# B&R Automation Studio project PloterCNC (part 3)

```c
/*****************************************************************************/
/* BEGIN: fmi2SerializeFMUstate */
/*****************************************************************************/
fmi2Status fmi2SerializeFMUstate(fmi2Component		c,
								fmi2FMUstate		FMUstate,
								fmi2Byte 			serializedState[],
								size_t				size) {
	ModelInstance* comp = (ModelInstance *)c;
	M_INT *icur;

	if (invalidState(comp, "fmi2SerializeFMUstate", modelInitialized))
		return fmi2Error;

	icur = (M_INT *)FMUstate;
	if(icur[0]!=FMUStateID) {
		compLog(compEnv, comp->instanceName, fmi2Error, "error",
			"fmi2SerializedFMUstate: called with invalid FMUstate");
		return fmi2Error;
	}
	if(icur[1]>(M_INT)size) {
		compLog(compEnv, comp->instanceName, fmi2Error, "error",
			"fmi2SerializedFMUstate: called with size not sufficient to contain FMUstate");
		return fmi2Error;
	}
	memcpy(serializedState, FMUstate, size);

	return fmi2OK;
}
/* END: fmi2SerializeFMUstate */
/*****************************************************************************/

/*****************************************************************************/
/* BEGIN: fmi2DeSerializeFMUstate */
/*****************************************************************************/
fmi2Status fmi2DeSerializeFMUstate(	fmi2Component	c,
									const fmi2Byte	serializedState[],
									size_t			size,
									fmi2FMUstate	*FMUstate) {
	ModelInstance* comp = (ModelInstance *)c;
	M_INT *icur;

	if (invalidState(comp, "fmi2DeSerializeFMUstate", modelInitialized))
		return fmi2Error;

	icur = (M_INT *)serializedState;
	if(icur[0]!=FMUStateID) {
		compLog(compEnv, comp->instanceName, fmi2Error, "error",
			"fmi2DeSerializedFMUstate: called with serializedState not containing valid FMUstate");
		return fmi2Error;
	}
	if(icur[1]>(M_INT)size) {
		compLog(compEnv, comp->instanceName, fmi2Error, "error",
			"fmi2SerializedFMUstate: called with size not sufficient to contain serializedState");
		return fmi2Error;
	}
	FMUstate[0] = (fmi2FMUstate)comp->functions.allocateMemory(1,size);
	memcpy(*FMUstate, serializedState, size);

	return fmi2OK;
}
/* END: fmi2DeSerializeFMUstate */
/*****************************************************************************/

/*****************************************************************************/
/* BEGIN: fmi2GetDirectionalDerivative */
/*****************************************************************************/
fmi2Status fmi2GetDirectionalDerivative(	fmi2Component			c,
										const fmi2ValueReference	vUnknown_ref[],
										size_t						nUnknown,
										const fmi2ValueReference	vKnown_ref[],
										size_t						nKnown,
										const fmi2Real				dvKnown[],
										fmi2Real					dvUnknown[]) {
#ifdef FMI2_PROVIDES_DERIVATIVES
	int i, j, k, row, col, offset;
	fmi2Status sts;
	fmi2ValueReference vrs, vrd;
	ModelInstance* comp = (ModelInstance *)c;

	if (invalidState(comp, "fmi2GetDirectionalDerivatives", modelInstantiated|modelInitialized))
		return fmi2Error;
	if (nKnown>0 && nullPointer(comp, "fmi2GetDirectionalDerivative", "vKnown_ref[]", vKnown_ref))
		return fmi2Error;
	if (nUnknown>0 && nullPointer(comp, "fmi2GetDirectionalDerivative", "vUnknown_ref[]", vUnknown_ref))
		return fmi2Error;
	if (nKnown>0 && nullPointer(comp, "fmi2GetDirectionalDerivative", "dvKnown[]", dvKnown))
		return fmi2Error;

	sts = syncModel(comp,"fmi2GetDirectionalDerivative");
	if ( sts!=fmi2OK ) return sts;

	/* Initialize unknown vector */
	for (i=0; i<nUnknown; i++) dvUnknown[i] = 0.;

	/* Get Jacobian information, dimensions, data, etc? */
	if(!comp->jsynced) {
		if(comp->initializeMode)
			initjac(comp->S.w[0],&(comp->S.w[1]),&(comp->S.w[NEQ+NPAR+1]),comp->initRes,comp->initJacobian);
		else
			intjac(comp->S.w[0],&(comp->S.w[1]),&(comp->S.w[NEQ+NPAR+1]),comp->Jacobian);
		comp->jsynced = fmi2True;
	}

	/* Order of value references :
	t, #states, #index-1(inps), #discrete, #params, #derivs, #events */

	/* Start the computation loop */
	if (comp->initializeMode) {
		offset = NIKNO;
		for (i=0; i<nKnown; i++) {
			/* Check the seed */
			if (dvKnown[i]!=0) {
				vrs = vKnown_ref[i];
				/* assert(vr>=0 && vr<NUMBER_OF_REALS); */
				col = -1;
				for (k=0; k<NIKNO; k++)
					if (vrs==vrIknowns[k]) {
						col = k;
						break;
					}
				/* Compute column i */
				for (j=0; j<nUnknown; j++) {
					vrd = vUnknown_ref[j];
					/* assert(vrd>=0 && vrd<NUMBER_OF_REALS); */
					if ( vrd==vrs ) {
						dvUnknown[j] += 1.0;
					}
					else if(col!=-1) {
						for (k=0; k<NIUNK; k++)
							if (vrd==vrIunknowns[k]) {
								dvUnknown[j] += dvKnown[i]*comp->initJacobian[k*offset+col];
								break;
							}
					}
				}
			}
		}
	}
	else {
		offset = 1+NDIFF+NINP;
		for (i=0; i<nKnown; i++) {
			/* Check the seed */
			if (dvKnown[i]!=0) {
				vrs = vKnown_ref[i];
				/* assert(vr>=0 && vr<NUMBER_OF_REALS); */
				/* Check that vKnown_ref[i] is a state or input */
				if ( vrs==0 || (vrs>=vrStates[0] && vrs<vrStates[0]+NDIFF) )
					col = vrs;
				else if(vrs>=1+NDIFF+NIX1-NINP && vrs<1+NDIFF+NIX1)
					col = vrs-(NIX1-NINP);
				else
					return fmi2Error;
				/* Compute column i */
				for (j=0; j<nUnknown; j++) {
					vrd = vUnknown_ref[j];
					/* assert(vrd>=0 && vrd<NUMBER_OF_REALS); */
					/* Check if vrd is a derivative or an output,
					it could also be an output that's a state */
					if ( vrd>=vrDers[0] && vrd<vrDers[0]+NDIFF ) {
						row = vrd-vrDers[0];
						dvUnknown[j] += dvKnown[i]*comp->Jacobian[row*offset+col];
					}
					else if( vrd>=vrStates[0] && vrd<vrStates[0]+NDIFF ) {
						if ( vrd==vrs ) dvUnknown[j] += 1.0;
					}
					else {
						for (k=0; k<NOUT; k++)
							if (vrd==vrOuts[k]) {
								/* refval-t-states+derivs: vrd-1-NDIFF+NDIFF */
								row = vrd-1;
								dvUnknown[j] += dvKnown[i]*comp->Jacobian[row*offset+col];
								break;
							}
						if (k==NOUT) return fmi2Error;
					}
				}
			}
		}
	}
	return fmi2OK;
#else
	/* Compiler warning fix */
	int i=nUnknown+nKnown;
	void *tmp;
	tmp=(void *)vUnknown_ref;
	tmp=(void *)vKnown_ref;
	tmp=(void *)dvKnown;
	tmp=(void *)dvUnknown;
	if(i>0) tmp=(void *)c;
	/* End compiler warning fix */
	return fmi2Error;
#endif
}
/* END: fmi2GetDirectionalDerivative */
/*****************************************************************************/

#if NCON>0 && defined(WMI_PROJECTION)
/*****************************************************************************/
/* BEGIN: fmi2Projection */
/*****************************************************************************/
fmi2Status fmi2Projection(	fmi2Component	c,
								fmi2Real	P[],
								fmi2Real	projectionTolerance,
								size_t	iterationLimit,
								fmi2Boolean	apply) {
	int i;
	fmi2Status sts;
	fmi2Real S2[NDIFF];

	ModelInstance* comp = (ModelInstance *)c;

	if (invalidState(comp, "fmi2Projection", modelInstantiated|modelInitialized))
		return fmi2Error;

	sts = syncModel(comp,"fmi2Projection");
	if ( sts!=fmi2OK ) return sts;

	for(i=0;i<NDIFF;i++) S2[i] = comp->S.w[i+1];
	i=Projection(comp->S.w[0], &comp->S.w[1], projectionTolerance, iterationLimit, NULL, comp->S.psto);
	if( i!=0 ){
		/* Restore state */
		for(i=0;i<NDIFF;i++) comp->S.w[i+1]=S2[i];
		return fmi2Discard;
	}
	for(i=0;i<NDIFF;i++) P[i] = comp->S.w[i+1]-S2[i];

	if( !apply ){
		for(i=0;i<NDIFF;i++) comp->S.w[i+1]=S2[i];
	}

	return fmi2OK;
}
/* END: fmi2Projection */
/*****************************************************************************/

/*****************************************************************************/
/* BEGIN: fmi2ProjectionStep: No longer supported */
/*****************************************************************************/
fmi2Status fmi2ProjectionStep(	fmi2Component	c,
									fmi2Real	S[]) {
	UNUSED(c);
	UNUSED(S);
		return fmi2Error;
}
/* END: fmi2ProjectionStep */
/*****************************************************************************/

/*****************************************************************************/
/* BEGIN: fmi2Constraint */
/*****************************************************************************/
fmi2Status fmi2Constraint(	fmi2Component	c,
								fmi2Real	C[]) {
	int cb, cr, nblk;
	fmi2Real blkdata[2];
	fmi2Status sts;

	ModelInstance* comp = (ModelInstance *)c;

	if (invalidState(comp, "fmi2Constraint", modelInstantiated|modelInitialized))
		return fmi2Error;

	sts = syncModel(comp,"fmi2Constraint");
	if ( sts!=fmi2OK ) return sts;

	/* Iterate over Residual blocks */
	Rblkp(comp->S.w[0], &comp->S.w[1], blkdata, 0, 0);
	nblk = (int)(blkdata[0]);
	cr = 0;
	for(cb=1;cb<=nblk;cb++) {
		Rblkp(comp->S.w[0], &comp->S.w[1], &C[cr], cb, 3);
		Rblkp(comp->S.w[0], &comp->S.w[1], blkdata, cb, 1);
		cr += (int)(blkdata[0]);
	}

	return fmi2OK;
}
/* END: fmi2Constraint*/
/*****************************************************************************/

/*****************************************************************************/
/* BEGIN: fmi2ConstraintJacobian: No longer supported */
/*****************************************************************************/
fmi2Status fmi2ConstraintJacobian(	fmi2Component	c,
										fmi2Real	J[]) {

	/* If this function is required at some point, the code will need to be
	modified to fill in the ncon x ndiff Matrix using a sequence of calls to
	the block-based Jacobian. It is known that this will provide 0 entries
	for block dependencies on vars from a prior block, but this will only
	slow convergence of a newton approach, and be irrelevant when sufficiently
	close to the solution manifold */
	UNUSED(c);
	UNUSED(J);
		return fmi2Error;
}
/* END: fmi2ConstraintJacobian*/
/*****************************************************************************/
#endif

#ifdef FMI2_COSIMULATION
/*****************************************************************************
 * FMI functions: only for FMI Co-Simulation 2.0
 *****************************************************************************/
/*****************************************************************************/
/* BEGIN: fmi2SetRealInputDerivatives */
fmi2Status fmi2SetRealInputDerivatives(	fmi2Component			c,
										const fmi2ValueReference vr[],
										size_t					nvr,
										const fmi2Integer		order[],
										const fmi2Real			value[]) {
	ModelInstance* comp = (ModelInstance *)c;

	if (invalidState(comp, "fmi2SetRealInputDerivatives", modelInitialized))
		return fmi2Error;
	if (comp->loggingOn)
		compLog(compEnv, comp->instanceName, fmi2OK, "log",
				"fmi2SetRealInputDerivatives: nvr= %d", nvr);

	compLog(NULL, comp->instanceName, fmi2Error, "warning",
			"fmi2SetRealInputDerivatives: ignoring function call."
			" This model cannot interpolate inputs: canInterpolateInputs = \"fmi2False\"");

	return fmi2Warning;
}
/* END: fmi2SetRealInputDerivatives */
/*****************************************************************************/

/*****************************************************************************/
/* BEGIN: fmi2GetRealOutputDerivatives */
fmi2Status fmi2GetRealOutputDerivatives(fmi2Component			c,
										const fmi2ValueReference vr[],
										size_t					nvr,
										const fmi2Integer		order[],
										fmi2Real				value[]) {
	int i;
	ModelInstance* comp = (ModelInstance *)c;

	if (invalidState(comp, "fmi2GetRealOutputDerivatives", modelInitialized))
		return fmi2Error;
	if (comp->loggingOn)
		compLog(compEnv, comp->instanceName, fmi2OK, "log",
				"fmi2GetRealOutputDerivatives: nvr= %d",	nvr);

	compLog(NULL, comp->instanceName, fmi2Error, "warning",
			"fmi2GetRealOutputDerivatives: ignoring function call."
			" This model cannot compute derivatives of outputs: MaxOutputDerivativeOrder=\"0\"");

	for (i=0; i<(int)nvr; i++) value[i] = 0;

	return fmi2Warning;
}
/* END: fmi2GetRealOutputDerivatives */
/*****************************************************************************/

#define MAX_STEP  1.00000000000000000e-03

/*****************************************************************************/
/* BEGIN: fmi2DoStep */
fmi2Status fmi2DoStep(  fmi2Component	c,
						fmi2Real		currentCommunicationPoint,
						fmi2Real		communicationStepSize,
						fmi2Boolean		newStep) {

	ModelInstance* comp	= (ModelInstance *)c;
	int		i;
	double	h;
	int		n;	/* how many internal steps to perform for one fmi2DoStep */
	int		k, hasEvent;
#if NEVT>0
	M_INT *modes;
	double	prevEventIndicators[max(NEVT, 1)], eventIndicators[max(NEVT, 1)];
#endif

	if (invalidState(comp, "fmi2DoStep", modelInitialized)) return fmi2Error;

	if (comp->loggingOn)
		compLog(compEnv, comp->instanceName, fmi2OK, "log", "fmi2DoStep: "
				"currentCommunicationPoint = %g, "
				"communicationStepSize = %g, "
				"newStep = fmi2%s",
				currentCommunicationPoint, communicationStepSize, newStep ? "True" : "False");

	if (comp->stopTimeDefined && currentCommunicationPoint+communicationStepSize > comp->stopTime) {
		comp->state = modelError;
		return fmi2Error;
	}

	if(communicationStepSize==0) {
		n = 1;
		h = 0.0;
	}
	else {
		n = (int)floor((communicationStepSize-1e-12)/MAX_STEP)+1;
		h = communicationStepSize/n;
	}

#if NPAR>0
	if(pchange) {
		SolverInitialize(&(comp->S));
		pchange=0;
		if (errorOccured>0) {
			setVidError(comp,NULL);
			if (comp->fptr) {
				writeErrorToFile(comp->fptr,NULL);
				comp->fptr = NULL;
			}
			comp->state = modelTerminated;
			logMessage(comp, "fmi2DoStep", "error", fmi2Error);
			return fmi2Error;
		}
		else if(errorOccured<0) {
			logMessage(comp, "fmi2DoStep", "warning", fmi2Warning);
			errorOccured=0;
		}
	}
#endif

#if NEVT>0
	/* Run to get initial event indicators */
	eev(comp->S.w[0],&(comp->S.w[1]),&(comp->S.w[1]),prevEventIndicators);
	modes=comp->S.iw;
	ComputeEventIndicators(prevEventIndicators,&(comp->S.w[1]),modes,
		&modes[3*NEVT],&modes[2*NEVT],&modes[4*NEVT]);
#endif

	comp->S.w[0] = currentCommunicationPoint;
	/* break the step into n steps and do a step */
	for (k=0; k<n; k++) {
#if NUMBER_OF_REALS>0
		if (h>0.0) {
			EulerStep(h,&(comp->S));
			if (errorOccured>0) {
				setVidError(comp,NULL);
				if (comp->fptr) {
					writeErrorToFile(comp->fptr,NULL);
					comp->fptr = NULL;
				}
				comp->state = modelTerminated;
				logMessage(comp,"EulerStep","error", fmi2Error);
				return fmi2Error;
			}
			else if(errorOccured<0) {
				logMessage(comp, "EulerStep", "warning", fmi2Warning);
				errorOccured=0;
			}
		}

		SolverUpdate(&(comp->S),0,1);
		if (errorOccured>0) {
			setVidError(comp,NULL);
			if (comp->fptr) {
				writeErrorToFile(comp->fptr,NULL);
				comp->fptr = NULL;
			}
			errorOccured = 0;
			comp->state = modelTerminated;
			logMessage(comp, "fmi2DoStep", "error", fmi2Discard);
			return fmi2Discard;
		}
		else if(errorOccured<0) {
			logMessage(comp, "fmi2DoStep", "warning", fmi2Warning);
			errorOccured=0;
		}
		comp->synced = fmi2True;
		comp->jsynced = fmi2False;

		i=SolverProject(&(comp->S));
		if(i<0 || errorOccured==1) {
			setVidError(comp,NULL);
			if (comp->fptr) {
				writeErrorToFile(comp->fptr,NULL);
				comp->fptr = NULL;
			}
			errorOccured = 0;
			comp->state = modelTerminated;
			logMessage(comp, "fmi2DoStep", "error", fmi2Error);
			return fmi2Error;
		}
		else if(i>0 || errorOccured==2) {
			compLog(compEnv, comp->instanceName, fmi2OK, "log",
					"fmi2DoStep: model requested termination at t = %g",
					comp->S.w[0]);
			setVidError(comp,NULL);
			if (comp->fptr) {
				writeErrorToFile(comp->fptr,NULL);
				comp->fptr = NULL;
			}
			errorOccured = 0;
			comp->state = modelTerminated;
			logMessage(comp, "fmi2DoStep", "warning", fmi2Discard);
			return fmi2Discard;
		}
		else if(errorOccured<0) {
			logMessage(comp, "fmi2DoStep", "warning", fmi2Warning);
			errorOccured=0;
		}
#endif
		hasEvent = 0;

#if NEVT>0
		/* check for state event */
		eev(comp->S.w[0],&(comp->S.w[1]),&(comp->S.w[1]),eventIndicators);
		modes=comp->S.iw;
		ComputeEventIndicators(eventIndicators,&(comp->S.w[1]),modes,
			&modes[3*NEVT],&modes[2*NEVT],&modes[4*NEVT]);
		for (i=0; i<NEVT; i++) {
			if (eventIndicators[i] * prevEventIndicators[i] < 0) {
				hasEvent = 1;
				if (comp->loggingOn)
					compLog(compEnv, comp->instanceName, fmi2OK, "log",
							"fmi2DoStep: state event at %g, z%d crosses zero -%c-",
							comp->S.w[0], i, eventIndicators[i]<0 ? '\\' : '/');
			}
			prevEventIndicators[i] = eventIndicators[i];
		}

		if (hasEvent) {
			i = RunEvents(comp->S.w, comp->S.iw, 0, -1, EVTITER, comp->S.psto);
			if (i>0 || errorOccured==2) {
				compLog(compEnv, comp->instanceName, fmi2OK, "log",
					"fmi2DoStep: model requested termination at t = %g",
					comp->S.w[0]);
			}
			else if (i<0 || errorOccured>0) {
				logMessage(comp, "fmi2DoStep", "error", fmi2Error);
			}
			if (i || errorOccured>0) {
				setVidError(comp,NULL);
				if (comp->fptr) {
					writeErrorToFile(comp->fptr,NULL);
					comp->fptr = NULL;
				}
				errorOccured = 0;
				comp->state = modelTerminated;
				return fmi2Discard;
			}
			if(errorOccured<0) {
				logMessage(comp, "fmi2DoStep", "warning", fmi2Warning);
				errorOccured=0;
			}
		}
#endif

		SolverOutputs(&(comp->S));
	}

	comp->lastSuccessfulTime = currentCommunicationPoint + communicationStepSize;
	comp->vidsts = 2;
 	if (comp->fptr)
		fwrite(comp->S.w,sizeof(fmi2Real),NEQ+1,comp->fptr);

	return fmi2OK;
}
/* END: fmi2DoStep */
/*****************************************************************************/

/*****************************************************************************/
/* BEGIN: fmi2CancelStep */
fmi2Status fmi2CancelStep(fmi2Component c) {
	ModelInstance* comp = (ModelInstance *)c;

	if (invalidState(comp, "fmi2CancelStep", modelInitialized)) return fmi2Error;
	if (comp->loggingOn)
		compLog(compEnv, comp->instanceName, fmi2OK, "log", "fmi2CancelStep");

	compLog(NULL, comp->instanceName, fmi2Error, "error",
			"fmi2CancelStep: Can be called when fmi2DoStep returned fmi2Pending."
			" This is not the case.");
	comp->state = modelError;
	return fmi2Error;
}
/* END: fmi2CancelStep */
/*****************************************************************************/

/*****************************************************************************/
/* BEGIN: fmi2GetStatus */
fmi2Status fmi2GetStatus(	fmi2Component		c,
							const fmi2StatusKind s,
							fmi2Status*			value) {
	ModelInstance* comp = (ModelInstance *)c;

	if (invalidState(comp, "fmi2GetStatus", modelInstantiated|modelInitialized))
		return fmi2Error;

	if (s==fmi2DoStepStatus) {
		if (comp->loggingOn) {
			compLog(compEnv, comp->instanceName, fmi2OK, "log",
				"[fmi2GetStatus]: fmi2StatusKind = fmi2DoStepStatus");
			compLog(NULL, comp->instanceName, fmi2Error, "error",
				"[fmi2GetStatus]: Can be called with fmi2DoStepStatus when fmi2DoStep returned fmi2Pending."
				" This is not the case.");
		}
		return fmi2Discard;
	}
	else
		return fmi2Discard;
}
/* END: fmi2GetStatus */
/*****************************************************************************/

/*****************************************************************************/
/* BEGIN: fmi2GetRealStatus */
fmi2Status fmi2GetRealStatus(	fmi2Component		c,
								const fmi2StatusKind s,
								fmi2Real*			value) {
	ModelInstance* comp = (ModelInstance *)c;

	if (invalidState(comp, "fmi2GetRealStatus", modelInstantiated|modelInitialized))
		return fmi2Discard;

	if (s==fmi2LastSuccessfulTime) {
		if (comp->loggingOn) {
			compLog(compEnv, comp->instanceName, fmi2OK, "log",
				"[fmi2GetRealStatus]: fmi2StatusKind = fmi2LastSuccessfulTime");
		}
		if (comp->state==modelTerminated) {
			*value = comp->lastSuccessfulTime;
			return fmi2OK;
		}
		else {
			compLog(NULL, comp->instanceName, fmi2Error, "error",
				"[fmi2GetRealStatus]: Can be called with fmi2LastSuccessfulTime when fmi2DoStep returned fmi2Discard."
				" This is not the case.");
			return fmi2Discard;
		}
	}
	else
		return fmi2Discard;
}
/* END: fmi2GetRealStatus */
/*****************************************************************************/

/*****************************************************************************/
/* BEGIN: fmi2GetIntegerStatus */
fmi2Status fmi2GetIntegerStatus(fmi2Component		c,
								const fmi2StatusKind s,
								fmi2Integer*		value) {
	return fmi2Discard;
}
/* END: fmi2GetIntegerStatus */
/*****************************************************************************/

/*****************************************************************************/
/* BEGIN: fmi2GetBooleanStatus */
fmi2Status fmi2GetBooleanStatus(fmi2Component		c,
								const fmi2StatusKind s,
								fmi2Boolean*		value) {
	ModelInstance* comp = (ModelInstance *)c;

	if (invalidState(comp, "fmi2GetBooleanStatus", modelInstantiated|modelInitialized))
		return fmi2Discard;

	if (s==fmi2Terminated) {
		if (comp->loggingOn) {
			compLog(compEnv, comp->instanceName, fmi2OK, "log",
				"[fmi2GetBooleanStatus]: fmi2StatusKind = fmi2Terminated");
		}
		if (comp->state==modelTerminated)
			*value = fmi2True;
		else
			*value = fmi2False;
		return fmi2OK;
	}
	else
		return fmi2Discard;
}
/* END: fmi2GetBooleanStatus */
/*****************************************************************************/

/*****************************************************************************/
/* BEGIN: fmi2GetStringStatus */
fmi2Status fmi2GetStringStatus(	fmi2Component		c,
								const fmi2StatusKind s,
								fmi2String*			value) {
	ModelInstance* comp = (ModelInstance *)c;

	if (invalidState(comp, "fmi2GetStringStatus", modelInstantiated|modelInitialized))
		return fmi2Discard;

	if (s==fmi2PendingStatus) {
		if (comp->loggingOn) {
			compLog(compEnv, comp->instanceName, fmi2OK, "log",
				"[fmi2GetStringStatus]: fmi2StatusKind = fmi2PendingStatus");
			compLog(NULL, comp->instanceName, fmi2Error, "error",
					"[fmi2GetStringStatus]: Can be called with fmi2PendingStatus when fmi2DoStep returned fmi2Pending."
					" This is not the case.");
		}
		return fmi2Discard;
	}
	else
		return fmi2Discard;
}
/* END: fmi2GetStringStatus */
/*****************************************************************************/

#else
/*****************************************************************************
 * FMI functions: only for Model Exchange 2.0
 *****************************************************************************/

/*****************************************************************************/
/* BEGIN: fmi2EnterEventMode */
fmi2Status fmi2EnterEventMode(fmi2Component c) {
	ModelInstance* comp = (ModelInstance *)c;

	if (comp) {
		comp->lastEventTime = comp->S.w[0]-1.0;
		return fmi2OK;
	}
	else
		return fmi2Error;
}
/* END: fmi2EnterEventMode */
/*****************************************************************************/

/*****************************************************************************/
/* BEGIN: fmi2NewDiscreteStates */
fmi2Status fmi2NewDiscreteStates(fmi2Component	c,
								fmi2EventInfo*	eventInfo) {
	ModelInstance* comp = (ModelInstance *)c;
	int i;
#if NEVT+NCON>0
	fmi2Real save[NEQ],val;
#endif
	if (invalidState(comp, "fmi2NewDiscreteStates", modelInitialized))
		return fmi2Error;
	if (nullPointer (comp, "fmi2NewDiscreteStates", "eventInfo", eventInfo))
		return fmi2Error;

	eventInfo->newDiscreteStatesNeeded				= fmi2False;
	eventInfo->nominalsOfContinuousStatesChanged	= fmi2False;
	eventInfo->valuesOfContinuousStatesChanged		= fmi2False;
	eventInfo->terminateSimulation					= fmi2False;
	eventInfo->nextEventTimeDefined					= fmi2False;
	eventInfo->nextEventTime						= -0.0;

#if NEVT+NCON>0
	for(i=0;i<NEQ;i++) save[i]=comp->S.w[i+1];
#endif
	i=SolverProject(&(comp->S));
	if (i<0 || errorOccured==1) {
		setVidError(comp,NULL);
		if (comp->fptr) {
			writeErrorToFile(comp->fptr,NULL);
			comp->fptr = NULL;
		}
		eventInfo->terminateSimulation = fmi2True;
		comp->state = modelTerminated;
		logMessage(comp, "fmi2NewDiscreteStates", "error", fmi2Error);
		return fmi2Error;
	}
	else if (i>0 || errorOccured==2) {
		compLog(compEnv, comp->instanceName, fmi2OK, "log",
				"fmi2NewDiscreteStates: model requested termination at t = %g",
				comp->S.w[0]);
		setVidError(comp,NULL);
		if (comp->fptr) {
			writeErrorToFile(comp->fptr,NULL);
			comp->fptr = NULL;
		}
		eventInfo->terminateSimulation = fmi2True;
		comp->state = modelTerminated;
		logMessage(comp, "fmi2NewDiscreteStates", "warning", fmi2Discard);
		return fmi2OK;
	}
	else if(errorOccured<0) {
		logMessage(comp, "fmi2NewDiscreteStates", "warning", fmi2Warning);
		errorOccured=0;
	}
#if NEVT>0
	if (comp->S.w[0]!=comp->lastEventTime) {
		i=RunEvents(comp->S.w, comp->S.iw, 0, -1, EVTITER, comp->S.psto);
		if (i<0 || errorOccured==1) {
			setVidError(comp,NULL);
			if (comp->fptr) {
				writeErrorToFile(comp->fptr,NULL);
				comp->fptr = NULL;
			}
			eventInfo->terminateSimulation = fmi2True;
			comp->state = modelTerminated;
			logMessage(comp, "fmi2NewDiscreteStates", "error", fmi2Error);
			return fmi2Error;
		}
		else if (i>0 || errorOccured==2) {
			compLog(compEnv, comp->instanceName, fmi2OK, "log",
					"fmi2NewDiscreteStates: model requested termination at t = %g",
					comp->S.w[0]);
			setVidError(comp,NULL);
			if (comp->fptr) {
				writeErrorToFile(comp->fptr,NULL);
				comp->fptr = NULL;
			}
			eventInfo->terminateSimulation = fmi2True;
			comp->state = modelTerminated;
			logMessage(comp, "fmi2NewDiscreteStates", "warning", fmi2Discard);
			return fmi2OK;
		}
		else if(errorOccured<0) {
			logMessage(comp, "fmi2NewDiscreteStates", "warning", fmi2Warning);
			errorOccured=0;
		}
		comp->lastEventTime = comp->S.w[0];
	}
	i=RunEvents(comp->S.w, comp->S.iw, 1, -1, EVTITER, comp->S.psto);
	if (i<0 || errorOccured==1) {
		setVidError(comp,NULL);
		if (comp->fptr) {
			writeErrorToFile(comp->fptr,NULL);
			comp->fptr = NULL;
		}
		eventInfo->terminateSimulation = fmi2True;
		comp->state = modelTerminated;
		logMessage(comp, "fmi2NewDiscreteStates", "error", fmi2Error);
		return fmi2Error;
	}
	else if (i>0 || errorOccured==2) {
		compLog(compEnv, comp->instanceName, fmi2OK, "log",
				"fmi2NewDiscreteStates: model requested termination at t = %g",
				comp->S.w[0]);
		setVidError(comp,NULL);
		if (comp->fptr) {
			writeErrorToFile(comp->fptr,NULL);
			comp->fptr = NULL;
		}
		eventInfo->terminateSimulation = fmi2True;
		comp->state = modelTerminated;
		logMessage(comp, "fmi2NewDiscreteStates", "warning", fmi2Discard);
		return fmi2OK;
	}
	else if(errorOccured<0) {
		logMessage(comp, "fmi2NewDiscreteStates", "warning", fmi2Warning);
		errorOccured=0;
	}
#endif
#if NEVT+NCON>0
	for(i=0;i<NEQ;i++) {
		val=1e-15;
		if(fabs(save[i])>val) val=fabs(save[i]);
		if(fabs(comp->S.w[i+1])>val) val=fabs(comp->S.w[i+1]);
		if( fabs(comp->S.w[i+1]-save[i])>1e-12*val )
			eventInfo->valuesOfContinuousStatesChanged = fmi2True;
	}
	if(eventInfo->valuesOfContinuousStatesChanged==fmi2True)
		SolverOutputs(&(comp->S));
#endif
	return fmi2OK;
}
/* END: fmi2NewDiscreteStates */
/*****************************************************************************/

/*****************************************************************************/
/* BEGIN: fmi2EnterContinuousTimeMode */
fmi2Status fmi2EnterContinuousTimeMode(fmi2Component c) {
	if (c)	return fmi2OK;
	else	return fmi2Error;
}
/* END: fmi2EnterContinuousTimeMode */
/*****************************************************************************/

/*****************************************************************************/
/* BEGIN: fmi2CompletedIntegratorStep */
fmi2Status fmi2CompletedIntegratorStep(	fmi2Component	c,
										fmi2Boolean		noSetFMUStatePriorToCurrentPoint,
										fmi2Boolean*	enterEventMode,
										fmi2Boolean*	terminateSimulation) {
	ModelInstance* comp = (ModelInstance *)c;
	int i;
#if NCON>0 && defined(CONDSTEPEVENT)
	fmi2Real save[NEQ],val,drift;
#endif

	UNUSED(noSetFMUStatePriorToCurrentPoint);
	if (invalidState(comp, "fmi2CompletedIntegratorStep", modelInitialized))
		return fmi2Error;
	if (nullPointer (comp, "fmi2CompletedIntegratorStep", "enterEventMode", enterEventMode))
		return fmi2Error;
	if (nullPointer (comp, "fmi2CompletedIntegratorStep", "terminateSimulation", terminateSimulation))
		return fmi2Error;
	if (comp->loggingOn)
		compLog(compEnv, comp->instanceName, fmi2OK, "log",
				"fmi2CompletedIntegratorStep");

	*terminateSimulation = fmi2False;

	if (comp->synced)
		SolverUpdate(&(comp->S),1,1);
	else {
		SolverUpdate(&(comp->S),0,1);
		if (errorOccured>0) {
			setVidError(comp,NULL);
			if (comp->fptr) {
				writeErrorToFile(comp->fptr,NULL);
				comp->fptr = NULL;
			}
			errorOccured = 0;
			comp->state = modelTerminated;
			logMessage(comp, "fmi2CompletedIntegratorStep", "error", fmi2Discard);
			return fmi2Discard;
		}
		else if(errorOccured<0) {
			logMessage(comp, "fmi2CompletedIntegratorStep", "warning", fmi2Warning);
			errorOccured=0;
		}
		comp->synced = fmi2True;
		comp->jsynced = fmi2False;
	}
	if(comp->fmuType==fmi2ModelExchange && comp->S.wset)
		for(i=NDIFF+1;i<=NDIFF+NIX1-NINP;i++)
			comp->S.wset[i]=comp->S.w[i];
	SolverOutputs(&(comp->S));
	if( comp->S.w[0]>=(comp->vidlasttime+comp->minSampleStep)*(1-1e-15) ) {
		comp->vidsts=2;
		comp->vidlasttime=comp->S.w[0];
	}
 	if (comp->fptr)
		if ( comp->S.w[0]>=(comp->lastsampletime+comp->minSampleStep)*(1-1e-15) ) {
			fwrite(comp->S.w,sizeof(fmi2Real),NEQ+1,comp->fptr);
			comp->lastsampletime=comp->S.w[0];
			if ( comp->numpts++ == WARNNUMDATPTS )
				compLog(compEnv, comp->instanceName, fmi2Warning, "warning",
						"[fmi2CompletedIntegratorStep]: At time t=%.16g, %d data points were written into file %s; consider increasing the minimum sample step, %.16g, to limit file size.",
						comp->S.w[0], WARNNUMDATPTS, comp->fstr, comp->minSampleStep);
		}

#if !defined(WMI_PROJECTION) && NCON>0
#   if defined(CONDSTEPEVENT)
	for(i=0;i<NEQ;i++) save[i]=comp->S.w[i+1];
	i=SolverProject(&(comp->S));
	if (i<0 || errorOccured>=1) {
		errorOccured=0;
		*enterEventMode = fmi2True;
	}
	else if (i>0) {
		setVidError(comp,NULL);
		if (comp->fptr) {
			writeErrorToFile(comp->fptr,NULL);
			comp->fptr = NULL;
		}
		comp->state = modelTerminated;
		*terminateSimulation = fmi2True;
		logMessage(comp, "fmi2CompletedIntegratorStep", "error", fmi2Discard);
		return fmi2OK;
	}
	else {
		drift=0.0;
		for(i=0;i<NEQ;i++) {
			val=1e-15;
			if(fabs(save[i])>val) val=fabs(save[i]);
			if(fabs(comp->S.w[i+1])>val) val=fabs(comp->S.w[i+1]);
			val=fabs(comp->S.w[i+1]-save[i])/val;
			if(val>drift) drift=val;
		}
		val=(CONTOL<1e-8) ? 1e-10 : 0.01*CONTOL;
		if(drift>val)
			*enterEventMode = fmi2True;
		else
			*enterEventMode = fmi2False;
	}
	for(i=0;i<NEQ;i++) comp->S.w[i+1]=save[i];
#   else
	*enterEventMode = fmi2True;
#   endif
#else
	*enterEventMode = fmi2False;
#endif

	return fmi2OK;
}
/* END: fmi2CompletedIntegratorStep */
/*****************************************************************************/

/*****************************************************************************/
/* BEGIN: fmi2SetTime */
fmi2Status fmi2SetTime(	fmi2Component	c,
						fmi2Real		time) {
	ModelInstance* comp = (ModelInstance *)c;
	if (invalidState(comp, "fmi2SetTime", modelInstantiated|modelInitialized))
		return fmi2Error;
	if (comp->loggingOn)
		compLog(compEnv, comp->instanceName, fmi2OK, "log",
				"fmi2SetTime: time = %.16g", time);
	if (comp->S.w[0] != time) {
		comp->S.w[0] = time;
		comp->synced = fmi2False;
		comp->jsynced = fmi2False;
	}
	return fmi2OK;
}
/* END: fmi2SetTime */
/*****************************************************************************/

/*****************************************************************************/
/* BEGIN: fmi2SetContinuousStates */
fmi2Status fmi2SetContinuousStates(	fmi2Component	c,
									const fmi2Real	x[],
									size_t			nx){
	ModelInstance* comp = (ModelInstance *)c;
#if NDIFF>0
	double scalev;
	int i;
	fmi2ValueReference vr;
#endif

	if (invalidState (comp, "fmi2SetContinuousStates", modelInitialized))
		return fmi2Error;
	if (invalidNumber(comp, "fmi2SetContinuousStates", "nx", nx, NDIFF))
		return fmi2Error;
#if NDIFF>0
	if (nullPointer  (comp, "fmi2SetContinuousStates", "x[]", x))
		return fmi2Error;

	for (i=0; i<(int)nx; i++) {
		vr = vrStates[i];
		if (comp->loggingOn)
			compLog(compEnv, comp->instanceName, fmi2OK, "log",
					"fmi2SetContinuousStates: #r%d# = %.16g", vr, x[i]);
		/*assert(vr>=0 && vr<NUMBER_OF_REALS);*/
		if( nomfac )
			scalev = nomfac[i]*x[i];
		else
			scalev = x[i];
		if (comp->S.w[vr] != scalev) {
			comp->S.w[vr] = scalev;
			comp->synced = fmi2False;
			comp->jsynced = fmi2False;
		}
	}
#endif
	return fmi2OK;
}
/* END: fmi2SetContinuousStates */
/*****************************************************************************/

/*****************************************************************************/
/* BEGIN: fmi2GetDerivatives */
fmi2Status fmi2GetDerivatives(	fmi2Component	c,
								fmi2Real		derivatives[],
								size_t			nx) {
#if NDIFF>0
	int i;
#endif
	ModelInstance* comp = (ModelInstance *)c;

	if (invalidState (comp, "fmi2GetDerivatives", validGet))
		return fmi2Error;
	if (invalidNumber(comp, "fmi2GetDerivatives", "nx", nx, NDIFF))
		return fmi2Error;
	if (nullPointer  (comp, "fmi2GetDerivatives", "derivatives[]", derivatives))
		return fmi2Error;

#if NDIFF>0
	if (comp->state==modelInitialized && !comp->synced) {
		SolverUpdate(&(comp->S),0,0);
		if(errorOccured>0) {
			setVidError(comp,NULL);
			if (comp->fptr) {
				writeErrorToFile(comp->fptr,NULL);
				comp->fptr = NULL;
			}
			errorOccured=0;
			logMessage(comp, "fmi2GetDerivatives", "error", fmi2Discard);
			return fmi2Discard;
		}
		else if(errorOccured<0) {
			logMessage(comp, "fmi2GetDerivatives", "warning", fmi2Warning);
			errorOccured=0;
		}
		comp->synced = fmi2True;
		comp->jsynced = fmi2False;
	}
	for (i=0; i<(int)nx; i++) {
		if( nomfac )
			derivatives[i] = comp->S.w[vrDers[i]]/nomfac[i];
		else
			derivatives[i] = comp->S.w[vrDers[i]];
		if (comp->loggingOn)
			compLog(compEnv, comp->instanceName, fmi2OK, "log",
					"fmi2GetDerivatives: #r%d# = %.16g",	vrDers[i], derivatives[i]);
	}
#endif
	return fmi2OK;
}
/* END: fmi2GetDerivatives */
/*****************************************************************************/

/*****************************************************************************/
/* BEGIN: fmi2GetEventIndicators */
fmi2Status fmi2GetEventIndicators(	fmi2Component	c,
									fmi2Real		eventIndicators[],
									size_t			ni) {
#if NEVT>0
	int i;
	M_INT *modes;
	fmi2Status sts;
#endif
	ModelInstance* comp = (ModelInstance *)c;

	if (invalidState (comp, "fmi2GetEventIndicators", validGet))
		return fmi2Error;
	if (invalidNumber(comp, "fmi2GetEventIndicators", "ni", ni, NEVT))
		return fmi2Error;

#if NEVT>0
	sts = syncModel(c,"fmi2GetEventIndicators");
	if ( sts!=fmi2OK ) return(sts);
	eev(comp->S.w[0],&(comp->S.w[1]),&(comp->S.w[1]),eventIndicators);
	modes=comp->S.iw;
	ComputeEventIndicators(eventIndicators,&(comp->S.w[1]),modes,
		&modes[3*NEVT],&modes[2*NEVT],&modes[4*NEVT]);
	for (i=0; i<(int)ni; i++) {
		if (comp->loggingOn)
			compLog(compEnv, comp->instanceName, fmi2OK, "log",
					"fmi2GetEventIndicators: z%d = %.16g",
					i, eventIndicators[i]);
	}
#else
	UNUSED(eventIndicators);
#endif
	return fmi2OK;
}
/* END: fmi2GetEventIndicators */
/*****************************************************************************/

/*****************************************************************************/
/* BEGIN: fmi2GetContinuousStates */
fmi2Status fmi2GetContinuousStates(	fmi2Component	c,
									fmi2Real		states[],
									size_t			nx) {
#if NDIFF>0
	int i;
	fmi2Status sts;
#endif
	ModelInstance* comp = (ModelInstance *)c;

	if (invalidState (comp, "fmi2GetContinuousStates", validGet))
		return fmi2Error;
	if (invalidNumber(comp, "fmi2GetContinuousStates", "nx", nx, NDIFF))
		return fmi2Error;
#if NDIFF>0
	if (nullPointer  (comp, "fmi2GetContinuousStates", "states[]", states))
		return fmi2Error;

	sts = syncModel(c,"fmi2GetContinuousStates");
	if ( sts!=fmi2OK ) return(sts);
	for (i=0; i<(int)nx; i++) {
		if( nomfac )
			states[i] = comp->S.w[vrStates[i]]/nomfac[i];
		else
			states[i] = comp->S.w[vrStates[i]];
		if (comp->loggingOn)
			compLog(compEnv, comp->instanceName, fmi2OK, "log",
					"fmi2GetContinuousStates: #r%u# = %.16g", vrStates[i], states[i]);
	}
#endif
	return fmi2OK;
}
/* END: fmi2GetContinuousStates */
/*****************************************************************************/

/*****************************************************************************/
/* BEGIN: fmi2GetNominalsOfContinuousStates */
fmi2Status fmi2GetNominalsOfContinuousStates(fmi2Component	c,
											fmi2Real		x_nominal[],
											size_t			nx) {
	ModelInstance* comp = (ModelInstance *)c;
	int i;

	if (invalidState (comp, "fmi2GetNominalsOfContinuousStates", validGet))
		return fmi2Error;
	if (invalidNumber(comp, "fmi2GetNominalsOfContinuousStates", "nx", nx, NDIFF))
		return fmi2Error;
	if (nullPointer  (comp, "fmi2GetNominalsOfContinuousStates", "x_nominal[]", x_nominal))
		return fmi2Error;

	if (comp->loggingOn)
		compLog(compEnv, comp->instanceName, fmi2OK, "log",
				"fmi2GetNominalsOfContinuousStates: x_nominal[0..%d] = 1.0", nx-1);
	if( nomfac )
		for (i=0; i<(int)nx; i++) x_nominal[i] = 1.0/nomfac[i-1];
	else
		for (i=0; i<(int)nx; i++) x_nominal[i] = 1.0;

	return fmi2OK;
}
/* END: fmi2GetNominalsOfContinuousStates */
/*****************************************************************************/

#endif

/*****************************************************************************/
/* Special purpose data communication functions */

typedef fmi2Status getMapleSimVideoDataLengthTYPE(fmi2Component, fmi2Integer *);
#define getMapleSimVideoDataLength fmi2FullName(getMapleSimVideoDataLength)
FMI2_Export getMapleSimVideoDataLengthTYPE getMapleSimVideoDataLength;

fmi2Status getMapleSimVideoDataLength(fmi2Component c, fmi2Integer *len)
{
	ModelInstance* comp = (ModelInstance *)c;

	if(comp->vidsts==0) {
		*len=0;
		return(fmi2Warning);
	}
	else if(comp->vidsts==1)
		*len=2+NPAR;
	else if(comp->vidsts==2)
		*len=NEQ+1;
	else if(comp->vidsts==-1)
		*len=2+strlen(comp->viderror)/8;
	else {
		*len=0;
		return(fmi2Error);
	}
	return(fmi2OK);
}

typedef fmi2Status getMapleSimVideoDataTYPE(fmi2Component, fmi2Real *);
#define getMapleSimVideoData fmi2FullName(getMapleSimVideoData)
FMI2_Export getMapleSimVideoDataTYPE getMapleSimVideoData;

fmi2Status getMapleSimVideoData(fmi2Component c, fmi2Real *data)
{
	ModelInstance* comp = (ModelInstance *)c;

	if(comp->vidsts==0)
		return(fmi2Error);
	else if(comp->vidsts==1) {
		data[0]=nData[0];
		data[1]=nData[1];
		memcpy(&data[2],&comp->S.w[NEQ+1],NPAR*sizeof(fmi2Real));
	}
	else if(comp->vidsts==2)
		memcpy(data,comp->S.w,(NEQ+1)*sizeof(fmi2Real));
	else if(comp->vidsts==-1) {
		data[0]=-1e10;
		memcpy(&data[1],comp->viderror,strlen(comp->viderror)+1);
	}
	else
		return(fmi2Error);
	comp->vidsts=0;
	return(fmi2OK);
}

typedef fmi2Status getMapleSimAuxiliaryDataTYPE(fmi2Component, fmi2Real *);
#define getMapleSimAuxiliaryData fmi2FullName(getMapleSimAuxiliaryData)
FMI2_Export getMapleSimAuxiliaryDataTYPE getMapleSimAuxiliaryData;

fmi2Status getMapleSimAuxiliaryData(fmi2Component c, fmi2Real *data)
{
	ModelInstance* comp = (ModelInstance *)c;

	if(!comp->synced) {
		auxp(comp->S.w[0],&(comp->S.w[1]),&(comp->S.w[NEQ+NPAR+1]),data);
		return(fmi2Discard);
	}
	else if(comp->state==modelInitialized) {
		auxp(comp->S.w[0],&(comp->S.w[1]),&(comp->S.w[NEQ+NPAR+1]),data);
		return(fmi2OK);
	}
	else return(fmi2Error);
}
```

#### MSpltrFmiSceneView.c
```c
#include <bur/plctypes.h>
#include <sys_lib.h>
#include "MSpltrLib.h"

#include <fmi2Functions.h>

#include <stdlib.h>
#include <stdio.h>
#include <string.h>
#include <math.h>

void MSpltrView(struct MSpltrView* fubInstance)
{
	if (fubInstance->Enable == 1) {

		if (fubInstance->InstRef->Fmi2.Enabled) {
			MSpltr_getMapleSimAuxiliaryData(fubInstance->InstRef->Fmi2.Instance, &(fubInstance->vInternal));
		}

		int i;
		for (i=0; i <= 18; i++) {
			fubInstance->ObjPos[i] = (float)fubInstance->vInternal[i];
		}

		} else {

	}

}
```

#### MSpltrImpl.c
```c
/********************************************************************
 * COPYRIGHT -- Bernecker + Rainer
 ********************************************************************

 ********************************************************************
 * Basic fmu/fub implementation
 ********************************************************************/

#include <bur/plctypes.h>
#include <sys_lib.h>
#include <fmi2Functions.h>

#ifdef __cplusplus
	extern "C"
	{
#endif
#include "MSpltrLib.h"
#ifdef __cplusplus
	};
#endif

/**********************************************************************/
/* FUB interface declarations */
#define  FMU_Enable 			fubInstance->Enable

#define  FMU_Instance 			fubInstance->Internal.Fmi2.Instance
#define  FMU_Enabled 			fubInstance->Internal.Fmi2.Enabled
#define  FMU_Error 			fubInstance->Internal.Fmi2.Error
#define  FMU_EndTime    		fubInstance->Internal.Fmi2.EndTime
#define  FMU_StartTime    		fubInstance->Internal.Fmi2.StartTime
#define  FMU_CurrentTime   		fubInstance->Internal.Fmi2.CurrentTime
#define  FMU_StepSize    		fubInstance->Internal.Fmi2.StepSize
#define  FMU_Callbacks   		fubInstance->Internal.Fmi2.Callbacks

/**********************************************************************/
/* Method delcarations */
void MSpltr_fmuLogger(fmi2Component c, fmi2String instanceName, fmi2Status status, fmi2String category, fmi2String message, ...);
void* MSpltr_AllocateMemory(UDINT numElements, UDINT elementSize);
void MSpltr_FreeMemory(void* pMemory);

void MSpltr_initFMU(struct MSpltr* fubInstance);

void MSpltr_initFMUCallbacks(struct MSpltr* fubInstance);
void MSpltr_initFMUCoSimParameters(struct MSpltr* fubInstance);

void MSpltr_stepFMU(struct MSpltr* fubInstance);
void MSpltr_resetFMU (struct MSpltr* fubInstance);

void MSpltr_copyOutputsFromFmu(struct MSpltr* fubInstance);
void MSpltr_copyInputsToFmu(struct MSpltr* fubInstance);
void MSpltr_clearFmuOutputs(struct MSpltr* fubInstance);

/**********************************************************************/
/* FUB implementation */
void MSpltr(struct MSpltr* fubInstance)
{
	MSpltr_ProcessFmuState(fubInstance);
}

/* Processes the fmu states */
void  MSpltr_ProcessFmuState(struct MSpltr* fubInstance)
{
	if (FMU_Enable)
	{
		if (!FMU_Enabled)
		{
			MSpltr_initFMU(fubInstance);
			FMU_Enabled = fmi2True;
		}

		if(FMU_Error == 0)
		{
			MSpltr_stepFMU(fubInstance);
		}
	}else
	{
		if (FMU_Enabled)
		{
			MSpltr_resetFMU(fubInstance);
			FMU_Enabled = fmi2False;
		}
	}
	fubInstance->InstRef = &(fubInstance->Internal);
}

/* Initialises the FMU */
void MSpltr_initFMU(struct MSpltr* fubInstance)
{
	fmi2Status retStatus = fmi2OK;
	FMU_Error = 0;

	MSpltr_initFMUCoSimParameters(fubInstance);

	MSpltr_initFMUCallbacks(fubInstance);

	FMU_Instance = MSpltr_fmi2Instantiate("MSpltr",fmi2CoSimulation,"{d25602c7-833a-5e8d-e356-ec0e85f22cec}",NULL,&FMU_Callbacks,fmi2False,fmi2False);

	if (!FMU_Instance)
	{
		FMU_Error = fmi2True;
	}else
	{
		retStatus = MSpltr_fmi2SetupExperiment(FMU_Instance,0 ,0.0, FMU_StartTime, 0, FMU_EndTime);

		if (retStatus > fmi2Warning)
		{
			FMU_Error = fmi2True;
			return;
		}

		retStatus = MSpltr_fmi2EnterInitializationMode(FMU_Instance);
		if (retStatus > fmi2Warning)
		{
			FMU_Error = fmi2True;
			return;
		}

		retStatus = MSpltr_fmi2ExitInitializationMode(FMU_Instance);
		if (retStatus > fmi2Warning)
		{
			FMU_Error = fmi2True;
			return;
		}

		MSpltr_copyOutputsFromFmu(fubInstance);
	}
}

/* Initialize CoSimulation parmeters */
void MSpltr_initFMUCoSimParameters(struct MSpltr* fubInstance)
{
	FMU_StartTime = 0.00000000000000000e+00;
	FMU_EndTime = 0.0;
	FMU_StepSize = 1.00000000000000000e-03;

	FMU_CurrentTime = 0.0;
}

/* Initialize FMU callbacks */
void  MSpltr_initFMUCallbacks(struct MSpltr* fubInstance)
{
	FMU_Callbacks.Logger = MSpltr_fmuLogger;
	FMU_Callbacks.AllocateMemory = MSpltr_AllocateMemory;
	FMU_Callbacks.FreeMemory = MSpltr_FreeMemory;
	FMU_Callbacks.StepFinished = NULL;
	FMU_Callbacks.ComponentEnvironment = NULL;
}

/* Execute FMU steps */
void MSpltr_stepFMU(struct MSpltr* fubInstance)
{

	if (FMU_Error == 0)
	{
		MSpltr_copyInputsToFmu(fubInstance);

		fmi2Status retStatus = MSpltr_fmi2DoStep(FMU_Instance, FMU_CurrentTime, FMU_StepSize, fmi2True);

		if(retStatus <= fmi2Warning)
		{
			MSpltr_copyOutputsFromFmu(fubInstance);

			FMU_CurrentTime += FMU_StepSize;
		}else
		{
			FMU_Error = fmi2True;
		}
	}
}

/* Reset the FMU */
void MSpltr_resetFMU (struct MSpltr* fubInstance)
{
	fmi2Status retStatus = MSpltr_fmi2Reset(FMU_Instance);

	if(retStatus <= fmi2Warning)
	{
		MSpltr_clearFmuOutputs(fubInstance);
		FMU_CurrentTime = 0;
	}else
	{
		FMU_Error = fmi2True;
	}
}

/* Log FMU calls */
void MSpltr_fmuLogger(void *componentEnvironment, fmi2String instanceName, fmi2Status status, fmi2String category, fmi2String message, ...)
{

}

/* Allocate memory */
void* MSpltr_AllocateMemory(UDINT numElements, UDINT elementSize)
{
	void* address;
	UDINT status = 0;

	status = TMP_alloc(numElements * elementSize, &address);

	if (status == 0)
	{
		return address;
	}
	else
	{
		return NULL;
	}
}

/* Free allocated memory */
void MSpltr_FreeMemory(void* pMemory)
{
	free(pMemory);
}

/* Clear the output values of the FMU */
void MSpltr_clearFmuOutputs(struct MSpltr* fubInstance)
{
	/*Clear fmu output PositionX*/
	fubInstance->PositionX = 0.0;
	/*Clear fmu output PositionY*/
	fubInstance->PositionY = 0.0;
	/*Clear fmu output SpeedX*/
	fubInstance->SpeedX = 0.0;
	/*Clear fmu output SpeedY*/
	fubInstance->SpeedY = 0.0;
	/*Clear fmu output TorqueX*/
	fubInstance->TorqueX = 0.0;
	/*Clear fmu output TorqueY*/
	fubInstance->TorqueY = 0.0;

}

/* Copy output values from the FMU */
void MSpltr_copyOutputsFromFmu(struct MSpltr* fubInstance)
{
	fmi2ValueReference valueReference;
	fmi2Status retStatus = fmi2OK;

	/*Copy fmu output PositionX to PositionX */
	valueReference = 67;
	fmi2Real PositionX;
	retStatus = MSpltr_fmi2GetReal(FMU_Instance, &valueReference, 1, &PositionX);

	if(retStatus <= fmi2Warning)
	{
		fubInstance->PositionX = PositionX;
	}else
	{
		FMU_Error = fmi2True;
		return;
	}
	/*Copy fmu output PositionY to PositionY */
	valueReference = 68;
	fmi2Real PositionY;
	retStatus = MSpltr_fmi2GetReal(FMU_Instance, &valueReference, 1, &PositionY);

	if(retStatus <= fmi2Warning)
	{
		fubInstance->PositionY = PositionY;
	}else
	{
		FMU_Error = fmi2True;
		return;
	}
	/*Copy fmu output SpeedX to SpeedX */
	valueReference = 2;
	fmi2Real SpeedX;
	retStatus = MSpltr_fmi2GetReal(FMU_Instance, &valueReference, 1, &SpeedX);

	if(retStatus <= fmi2Warning)
	{
		fubInstance->SpeedX = SpeedX;
	}else
	{
		FMU_Error = fmi2True;
		return;
	}
	/*Copy fmu output SpeedY to SpeedY */
	valueReference = 4;
	fmi2Real SpeedY;
	retStatus = MSpltr_fmi2GetReal(FMU_Instance, &valueReference, 1, &SpeedY);

	if(retStatus <= fmi2Warning)
	{
		fubInstance->SpeedY = SpeedY;
	}else
	{
		FMU_Error = fmi2True;
		return;
	}
	/*Copy fmu output TorqueX to TorqueX */
	valueReference = 69;
	fmi2Real TorqueX;
	retStatus = MSpltr_fmi2GetReal(FMU_Instance, &valueReference, 1, &TorqueX);

	if(retStatus <= fmi2Warning)
	{
		fubInstance->TorqueX = TorqueX;
	}else
	{
		FMU_Error = fmi2True;
		return;
	}
	/*Copy fmu output TorqueY to TorqueY */
	valueReference = 70;
	fmi2Real TorqueY;
	retStatus = MSpltr_fmi2GetReal(FMU_Instance, &valueReference, 1, &TorqueY);

	if(retStatus <= fmi2Warning)
	{
		fubInstance->TorqueY = TorqueY;
	}else
	{
		FMU_Error = fmi2True;
		return;
	}
}

/* Copy input values to the FMU */
void MSpltr_copyInputsToFmu(struct MSpltr* fubInstance)
{
	fmi2ValueReference valueReference;
	fmi2Status retStatus = fmi2OK;

	/*Copy fmu input InputX to InputX */
	valueReference = 73;
	fmi2Real InputX;
	InputX = fubInstance->InputX;
	retStatus = MSpltr_fmi2SetReal(FMU_Instance, &valueReference, 1, &InputX);
	if(retStatus > fmi2Warning)
	{
		FMU_Error = fmi2True;
		return;
	}
	/*Copy fmu input InputY to InputY */
	valueReference = 74;
	fmi2Real InputY;
	InputY = fubInstance->InputY;
	retStatus = MSpltr_fmi2SetReal(FMU_Instance, &valueReference, 1, &InputY);
	if(retStatus > fmi2Warning)
	{
		FMU_Error = fmi2True;
		return;
	}
}
```

### Program Logical/MSpltrFmu/PloterCfg (IEC)

#### Variables.var
```iecst
VAR
	NewObjPos : ARRAY[0..18] OF REAL;
END_VAR
```

#### Main.st
```iecst
PROGRAM _INIT
	(* Insert code here *)

END_PROGRAM

PROGRAM _CYCLIC

	MSpltr1.Enable:=TRUE;
	MSpltrView_0.Enable:=TRUE;

	// input- velocity
	MSpltr1.InputX := MpAxisBasicX.Velocity*19;
	MSpltr1.InputY := -MpAxisBasicY.Velocity*19;

	MSpltr1();

	MSpltrView_0.InstRef := MSpltr1.InstRef;

	MSpltrView_0();

	gPozycjaX := MSpltr1.PositionX*10;
	gPozycjaY := MSpltr1.PositionY*10-420;

	// output- torque
	gTorqueX := MSpltr1.TorqueX*0.15;
	gTorqueY := MSpltr1.TorqueY*(-0.1);

	// offset
	brsmemcpy(ADR(NewObjPos), ADR(MSpltrView_0.ObjPos), SIZEOF(MSpltrView_0.ObjPos));
	NewObjPos[6] := MSpltrView_0.ObjPos[6]+439.53;
	// NewObjPos[] is used in Scene Viewer (PVI)

END_PROGRAM

PROGRAM _EXIT
	(* Insert code here *)

END_PROGRAM
```

### Program Logical/Programs/CNC_Programs/ManualContr (IEC)

#### Main.st - Init, cyclic, exit code
```iecst
PROGRAM _INIT

	gStartValueChanging;
	MpCnc2Axis_0;
	CncParameters;
	gActiveTool;

	gMoveAbsoluteX:=TRUE;
	gMoveAbsoluteY:=TRUE;

END_PROGRAM

PROGRAM _CYCLIC

	IF gManualContr OR ButtonEnable=FALSE THEN
		gAutomaticContr:=FALSE;
	ELSE
		gAutomaticContr:=TRUE;
	END_IF;

	IF MpCnc2Axis_0.MoveProgram THEN
	  gManualContr:=FALSE;
	END_IF;

	(*When activating manual control*)
	IF EDGEPOS(gManualContr) THEN
	MpBasicParametersX.Position:=MpCnc2Axis_0.X;
	MpBasicParametersY.Position:=MpCnc2Axis_0.Y;
	END_IF

	(*Manual control operating mode switched on with a button in Visu*)
	IF gManualContr THEN

		(*Movement controlled by sliders and text input in visualization*)

		PosX:=LREAL_TO_INT(MpBasicParametersX.Position);
		PosY:=LREAL_TO_INT(MpBasicParametersY.Position);

		IF MpBasicParametersX.Position=INT_TO_LREAL(CncPosX) THEN
			gMoveAbsoluteX:=FALSE;
		END_IF;

		IF MpBasicParametersY.Position=INT_TO_LREAL(CncPosY) THEN
			gMoveAbsoluteY:=FALSE;
		END_IF;

		(*Movement in X (MOVE ABSOLUTE) *)
		IF gMoveAbsoluteX THEN
			MpAxisBasicX.MoveAbsolute:=TRUE;
		END_IF;

		IF MpAxisBasicX.MoveDone=TRUE THEN
			MpAxisBasicX.MoveAbsolute:=FALSE;
			gMoveAbsoluteX:=FALSE;
		END_IF;

		IF EDGENEG(gMoveAbsoluteX) AND CncPosX<>PosX THEN
			gMoveAbsoluteX:=TRUE;
		END_IF;

		(*Movement in Y  (MOVE ABSOLUTE) *)

		IF gMoveAbsoluteY THEN
			MpAxisBasicY.MoveAbsolute:=TRUE;
		END_IF;

		IF MpAxisBasicY.MoveDone=TRUE THEN
			MpAxisBasicY.MoveAbsolute:=FALSE;
			gMoveAbsoluteY:=FALSE;
		END_IF;

		IF EDGENEG(gMoveAbsoluteY) AND CncPosY<>PosY THEN
			gMoveAbsoluteY:=TRUE;
		END_IF;

	ELSIF gManualContr=FALSE THEN
		MpAxisBasicX.MoveAbsolute:=FALSE;
		MpAxisBasicY.MoveAbsolute:=FALSE;
	END_IF;

	(*Movement control with ARROWS in visualization*)

	(*Arrows parameters*)

	MpBasicParametersX.Jog.Velocity:=gParameter.set_X_vel;
	MpBasicParametersY.Jog.Velocity:=gParameter.set_Z_vel;
	MpBasicParametersX.Jog.Acceleration:=gParameter.limit_acc;
	MpBasicParametersY.Jog.Acceleration:=gParameter.limit_acc;
	MpBasicParametersX.Jog.Deceleration:=gParameter.limit_dec;
	MpBasicParametersY.Jog.Deceleration:=gParameter.limit_dec;

	MpBasicParametersX.Jog.LimitPosition.FirstPosition:=0;
	MpBasicParametersX.Jog.LimitPosition.LastPosition:=520;
	MpBasicParametersY.Jog.LimitPosition.FirstPosition:=0;
	MpBasicParametersY.Jog.LimitPosition.LastPosition:=420;

	(*JOG MOVEMENT - NEGATIVE AND POSITIVE*)
	IF MpCnc2Axis_0.MoveActive AND (EDGENEG(MpAxisBasicX.JogNegative) OR EDGENEG(MpAxisBasicY.JogNegative) OR EDGENEG(MpAxisBasicX.JogPositive) OR EDGENEG(MpAxisBasicY.JogPositive)) THEN
	GetThere:=TRUE;
	END_IF;

	IF GetThere THEN
		MpBasicParametersY.Position:=MpCnc2Axis_0.Y;
		MpBasicParametersX.Position:=MpCnc2Axis_0.X;
	END_IF;

	IF MpCnc2Axis_0.MoveActive=FALSE THEN
		GetThere:=FALSE;
	END_IF

	(*Go Up, GoDown, GoLeft and GoRight are variables connected to the arrows in visu*)
	(*UP*)
	IF GoUp=TRUE THEN
		//	MpBasicParametersY.Position:=INT_TO_LREAL(CncPosY);
		MpBasicParametersY.Position:=MpCnc2Axis_0.Y;
		MpAxisBasicY.MoveAbsolute:=FALSE;
		MpAxisBasicY.JogNegative:=TRUE;

	ELSIF GoUp=FALSE THEN
		MpAxisBasicY.JogNegative:=FALSE;
	END_IF;

	(*DOWN*)
	IF GoDown THEN
		MpBasicParametersY.Position:=INT_TO_LREAL(CncPosY);
		MpAxisBasicY.MoveAbsolute:=FALSE;
		MpAxisBasicY.JogPositive:=TRUE;

	ELSIF GoDown=FALSE THEN
		MpAxisBasicY.JogPositive:=FALSE;
	END_IF;

	(*LEFT*)
	IF GoLeft  THEN
		MpBasicParametersX.Position:=INT_TO_LREAL(CncPosX);
		MpAxisBasicX.MoveAbsolute:=FALSE;
		MpAxisBasicX.JogNegative:=TRUE;

	ELSIF GoLeft=FALSE THEN
		MpAxisBasicX.JogNegative:=FALSE;
	END_IF;

		(*RIGHT*)
	IF GoRight THEN
		MpBasicParametersX.Position:=INT_TO_LREAL(CncPosX);
		MpAxisBasicX.MoveAbsolute:=FALSE;
		MpAxisBasicX.JogPositive:=TRUE;

	ELSIF GoRight=FALSE THEN
		MpAxisBasicX.JogPositive:=FALSE;
	END_IF;

	(*Limits for movement in both directions (x,y) *)

	IF MpBasicParametersY.Position>=420 THEN
		MpBasicParametersY.Position:=420;

	ELSIF MpBasicParametersY.Position<=0 THEN
		MpBasicParametersY.Position:=0;
	END_IF;

	IF MpBasicParametersX.Position>=520 THEN
		MpBasicParametersX.Position:=520;

	ELSIF MpBasicParametersX.Position<=0 THEN
		MpBasicParametersX.Position:=0;
	END_IF;

	(* A dot showing the position of the tool*)
	pointString:='<circle cx="';

	pointStrX:=REAL_TO_STRING(CncPosX*1.2);
	pointStrY:=REAL_TO_STRING(CncPosY*1.2);

	strHelp:='" cy="';
	strcat(ADR(pointString),ADR(pointStrX));
	strcat(ADR(pointString),ADR(strHelp));
	strcat(ADR(pointString),ADR(pointStrY));
	strHelp:='" r="5" stroke="black" stroke-width="3" fill="red" />';
	strcat(ADR(pointString),ADR(strHelp));

	MpAxisBasicX();
	MpAxisBasicY();

	IF MpAxisBasicX.Velocity=0 THEN
		gCurrentX:=0;
	ELSIF MpAxisBasicX.Velocity<0 THEN
		gCurrentX:=-MpAxisBasicX.Velocity*0.01+0.48;
	ELSIF MpAxisBasicX.Velocity>0 THEN
		gCurrentX:=MpAxisBasicX.Velocity*0.01+0.48;
		END_IF;

		IF MpAxisBasicY.Velocity=0 THEN
		gCurrentY:=0;
	ELSIF MpAxisBasicY.Velocity<0 THEN
		gCurrentY:=-MpAxisBasicY.Velocity*0.01+0.48;
	ELSIF MpAxisBasicY.Velocity>0 THEN
		gCurrentY:=MpAxisBasicY.Velocity*0.01+0.48;
		END_IF;

END_PROGRAM

PROGRAM _EXIT

END_PROGRAM
```

#### Variables.var - Local variables
```iecst
VAR
	PosY : INT;
	PosX : INT;
	GoDown : BOOL;
	GoRight : BOOL;
	GoLeft : BOOL;
	GoUp : BOOL;
	pointStrX : STRING[80];
	pointStrY : STRING[80];
	strHelp : STRING[80];
	pointString : STRING[120];
	GetThere : BOOL;
	gCurrentX : REAL;
	gCurrentY : REAL;
END_VAR
```

### Program Logical/Programs/live_drawing/live_draw

#### Variables.var
```iecst
VAR
	angle : REAL;
	cmdBack : BOOL;
	cmdClear : BOOL;
	cmdDraw : BOOL;
	curShape : shape_enum;
	i : UINT;
	InfoString : STRING[300];
END_VAR
VAR CONSTANT
	PI : REAL := 3.141592;
END_VAR
VAR
	prevReadX : UINT;
	prevReadY : UINT;
	radius : REAL := 100;
	PositionString : STRING[500];
	PositionArrayIndex : UINT;
	PositionArray : ARRAY[0..999] OF STRING[500];
	readX : UINT;
	readY : UINT;
	shapeString : STRING[500];
	smallRadius : REAL;
	stage : INT;
	strHelp : STRING[80];
	strPrevX : STRING[80];
	strPrevY : STRING[80];
	strRadius : STRING[80];
	strX : STRING[80];
	strY : STRING[80];
	svgStringArray : ARRAY[0..999] OF STRING[500];
	svgStringArrayIndex : UINT := 3;
	x : REAL;
	y : REAL;
	inXlinePosYStr : STRING[80];
	inXlinePosY : REAL;
	inXlinePosXStr : STRING[80];
	inXlinePosX : REAL;
	inXlinePosYStr1 : STRING[80];
	inXlinePosY1 : REAL;
	inYlinePosYStr : STRING[80];
	inYlinePosY : REAL;
	inYlinePosXStr : STRING[80];
	inYlinePosX : REAL;
	inYlinePosXStr1 : STRING[80];
	inYlinePosX1 : REAL;
	HelpLines : BOOL;
	readYRec : UINT := 40;
	readXRec : UINT := 40;
	strXRec : STRING[80];
	strYRec : STRING[80];
	CircleRadius : REAL := 70;
	strRot : STRING[80];
	RotationAngle : REAL;
	strPrevReadX : STRING[80];
	strPrevReadY : STRING[80];
	CurrentShape : STRING[80];
END_VAR
```

#### Main.st
```iecst
PROGRAM _INIT

	readX;
	readY;

END_PROGRAM

PROGRAM _CYCLIC

	(*Warning*)
	IF InfoString='Shape outside drawing field!' THEN
		gMsgBox:=TRUE;
	ELSE
		gMsgBox:=FALSE;
	END_IF;

	IF InfoString='Radius can not be equal to 0!' THEN
		gMsgBox2:=TRUE;
	ELSE
		gMsgBox2:=FALSE;
	END_IF;

	IF InfoString='Distance can not be equal to 0!' THEN
		gMsgBox3:=TRUE;
	ELSE
		gMsgBox3:=FALSE;
	END_IF;

	(*HelpLines*)
	IF HelpLines THEN

		IF (readX-inXlinePosX)<=20 AND (readY-inYlinePosY)<=20 AND (readY-inYlinePosY)>=-20 AND (readX-inXlinePosX)>=-20 THEN
			readX:=REAL_TO_UINT(inXlinePosX);
			readY:=REAL_TO_UINT(inYlinePosY);
		END_IF;

	END_IF;

	CASE curShape OF

		circle:

			CurrentShape:='circle';
			(*-circle drawing-*)
			CASE stage OF
				0:
			InfoString:='Point centre of the circle';
					IF EDGEPOS(cmdDraw) THEN
						cmdDraw:=FALSE;
						RotationAngle:=0;
						strRot:=REAL_TO_STRING(RotationAngle);
						shapeString:='<circle cx="';
						prevReadX:=readX;
						prevReadY:=readY;
						strX:=UINT_TO_STRING(readX);
						strY:=UINT_TO_STRING(readY);

						strHelp:='" cy="';
						strcat(ADR(shapeString),ADR(strX));
						strcat(ADR(shapeString),ADR(strHelp));
						strcat(ADR(shapeString),ADR(strY));
						strHelp:='" r="';
						strcat(ADR(shapeString),ADR(strHelp));
						stage:=1;

						IF prevReadX-CircleRadius<0 OR prevReadY-CircleRadius<0 OR prevReadX+CircleRadius>780 OR prevReadY+CircleRadius>630 THEN
							stage:=1;
						ELSIF CircleRadius=0 THEN
							stage:=2;
						ELSE
							strRadius:=REAL_TO_STRING(CircleRadius);
							strcat(ADR(shapeString),ADR(strRadius));
							strHelp:='" stroke="black" fill="none" />';
							strcat(ADR(shapeString),ADR(strHelp));

							svgStringArray[svgStringArrayIndex]:=shapeString;
							svgStringArrayIndex:=svgStringArrayIndex+1;

							IF svgStringArray[3]<>'' THEN

								(*PositionArray*)
								strHelp:='type:';
								strcat(ADR(PositionString), ADR(strHelp));
								strcat(ADR(PositionString), ADR(CurrentShape));
								strHelp:='; x=';
								strcat(ADR(PositionString), ADR(strHelp));

								strcat(ADR(PositionString), ADR(strX));
								strHelp:='; y=';
								strcat(ADR(PositionString), ADR(strHelp));
								strcat(ADR(PositionString), ADR(strY));;
								strHelp:='; rot=';
								strcat(ADR(PositionString), ADR(strHelp));
								strcat(ADR(PositionString), ADR(strRot));
								strHelp:='';
								strcat(ADR(PositionString), ADR(strHelp));

								PositionArray[PositionArrayIndex]:=PositionString;
								PositionArrayIndex:=PositionArrayIndex+1;
								PositionString:='';

							END_IF;

							stage:=0;

						END_IF;
					END_IF;

				1:
					InfoString:='Shape outside drawing field!';

					IF EDGEPOS(cmdDraw) THEN
						cmdDraw:=FALSE;
						stage:=0;
					END_IF;

				2:
					InfoString:='Radius can not be equal to 0!';
					IF EDGEPOS(cmdDraw) THEN
						cmdDraw:=FALSE;
						stage:=0;
					END_IF;

			END_CASE;

			(*---------------*)
		line:
			(*-line drawing-*)
			CASE stage OF

				0:
					CurrentShape:='line';

					InfoString:='Point first-point of the line';
					IF EDGEPOS(cmdDraw) THEN
						cmdDraw:=FALSE;
						shapeString:='<polyline points="';
						prevReadX:=readX;
						prevReadY:=readY;

						stage:=1;
					END_IF;

				1:
			InfoString:='Point end-point of the line';
					IF EDGEPOS(cmdDraw) THEN
						cmdDraw:=FALSE;
						strPrevX:=UINT_TO_STRING(prevReadX);
						strPrevY:=UINT_TO_STRING(prevReadY);
						strX:=UINT_TO_STRING(readX);
						strY:=UINT_TO_STRING(readY);
						strHelp:=',';
						strcat(ADR(shapeString),ADR(strPrevX));
						strcat(ADR(shapeString),ADR(strHelp));
						strcat(ADR(shapeString),ADR(strPrevY));
						strHelp:=' ';
						strcat(ADR(shapeString),ADR(strHelp));
						strHelp:=',';
						strcat(ADR(shapeString),ADR(strX));
						strcat(ADR(shapeString),ADR(strHelp));
						strcat(ADR(shapeString),ADR(strY));

						strHelp:='" fill="none" stroke="black" />';
						strcat(ADR(shapeString),ADR(strHelp));
						svgStringArray[svgStringArrayIndex]:=shapeString;

						svgStringArrayIndex:=svgStringArrayIndex+1;

						stage:=0;
					END_IF;

			END_CASE;

		(*---------------*)

		rectangle:
			(*-rectangle drawing-*)
			CurrentShape:='rectangle';
			CASE stage OF
				0:
			InfoString:='Point top-left corner of the rectangle';
					IF EDGEPOS(cmdDraw) THEN
						cmdDraw:=FALSE;
						shapeString:='<polyline points="';
						prevReadX:=readX;
						prevReadY:=readY;
						strPrevReadX:=UINT_TO_STRING(prevReadX);
						strPrevReadY:=UINT_TO_STRING(prevReadY);
						strRot:=REAL_TO_STRING(RotationAngle);

						IF prevReadX+readXRec>780 OR prevReadY+readYRec>630 THEN
							cmdDraw:=FALSE;
							stage:=1;
						ELSIF readXRec=0 OR readYRec=0 THEN
							stage:=2;
						ELSE
							strPrevX:=UINT_TO_STRING(prevReadX);
							strPrevY:=UINT_TO_STRING(prevReadY);
							strXRec:=UINT_TO_STRING(prevReadX+readXRec);
							strYRec:=UINT_TO_STRING(prevReadY+readYRec);
							strHelp:=',';
							strcat(ADR(shapeString),ADR(strPrevX));
							strcat(ADR(shapeString),ADR(strHelp));
							strcat(ADR(shapeString),ADR(strPrevY));
							strHelp:=' ';
							strcat(ADR(shapeString),ADR(strHelp));
							strHelp:=',';
							strcat(ADR(shapeString),ADR(strXRec));
							strcat(ADR(shapeString),ADR(strHelp));
							strcat(ADR(shapeString),ADR(strPrevY));
							strHelp:=' ';
							strcat(ADR(shapeString),ADR(strHelp));
							strHelp:=',';
							strcat(ADR(shapeString),ADR(strXRec));
							strcat(ADR(shapeString),ADR(strHelp));
							strcat(ADR(shapeString),ADR(strYRec));
							strHelp:=' ';
							strcat(ADR(shapeString),ADR(strHelp));
							strHelp:=',';
							strcat(ADR(shapeString),ADR(strPrevX));
							strcat(ADR(shapeString),ADR(strHelp));
							strcat(ADR(shapeString),ADR(strYRec));

							strHelp:=' ';
							strcat(ADR(shapeString),ADR(strHelp));
							strHelp:=',';
							strcat(ADR(shapeString),ADR(strPrevX));
							strcat(ADR(shapeString),ADR(strHelp));
							strcat(ADR(shapeString),ADR(strPrevY));
							strHelp:='" transform="rotate(';
							strcat(ADR(shapeString),ADR(strHelp));
							strcat(ADR(shapeString),ADR(strRot));
							strHelp:=' ';
							strcat(ADR(shapeString),ADR(strHelp));
							strcat(ADR(shapeString),ADR(strPrevX));
							strHelp:=',';
							strcat(ADR(shapeString),ADR(strHelp));
							strcat(ADR(shapeString),ADR(strPrevY));
							strHelp:=')"';
							strcat(ADR(shapeString),ADR(strHelp));
							strHelp:=' fill="none" stroke="black" />';
							strcat(ADR(shapeString),ADR(strHelp));
							svgStringArray[svgStringArrayIndex]:=shapeString;

							svgStringArrayIndex:=svgStringArrayIndex+1;

							IF svgStringArray[3]<>'' THEN

								(*PositionArray*)
								strHelp:='type:';
								strcat(ADR(PositionString), ADR(strHelp));
								strcat(ADR(PositionString), ADR(CurrentShape));
								strHelp:='; x=';
								strcat(ADR(PositionString), ADR(strHelp));
								strcat(ADR(PositionString), ADR(strPrevReadX));
								strHelp:='; y=';
								strcat(ADR(PositionString), ADR(strHelp));
								strcat(ADR(PositionString), ADR(strPrevReadY));
								strHelp:='; rot=';
								strcat(ADR(PositionString), ADR(strHelp));
								strcat(ADR(PositionString), ADR(strRot));
								strHelp:='';
								strcat(ADR(PositionString), ADR(strHelp));

								PositionArray[PositionArrayIndex]:=PositionString;
								PositionArrayIndex:=PositionArrayIndex+1;
								PositionString:='';
							END_IF;

							stage:=0;
						END_IF;
					END_IF;

				1:
					InfoString:='Shape outside drawing field!';

					IF EDGEPOS(cmdDraw) THEN
						cmdDraw:=FALSE;
						stage:=0;
					END_IF;

				2:
					InfoString:='Distance can not be equal to 0!';

					IF EDGEPOS(cmdDraw) THEN
						cmdDraw:=FALSE;
						stage:=0;
					END_IF;

			END_CASE;

		(*---------------*)

		star:
			(*-star drawing-*)
			CASE stage OF

				0:
					CurrentShape:='star';
					InfoString:='Point centre of the star';
					strRot:=REAL_TO_STRING(RotationAngle);

					IF EDGEPOS(cmdDraw) THEN
						cmdDraw:=FALSE;
						shapeString:='<polyline points="';
						prevReadX:=readX;
						prevReadY:=readY;
						strPrevReadX:=REAL_TO_STRING(prevReadX);
						strPrevReadY:=REAL_TO_STRING(prevReadY);
						cmdDraw:=FALSE;

						IF prevReadX-radius<0 OR prevReadY-radius<0 OR prevReadX+radius>780 OR prevReadY+radius>630 THEN
							stage:=1;
						ELSIF radius=0 THEN
							stage:=2;
						ELSE
							smallRadius:=radius/3;
							angle:=-18; // degrees
							FOR i:=1 TO 5 DO

								x:=radius*COS(angle/180*PI);
								y:=radius*SIN(angle/180*PI);
								strX:=REAL_TO_STRING(x+prevReadX);
								strY:=REAL_TO_STRING(y+prevReadY);
								strHelp:=',';
								strcat(ADR(shapeString),ADR(strX));
								strcat(ADR(shapeString),ADR(strHelp));
								strcat(ADR(shapeString),ADR(strY));
								strHelp:=' ';
								strcat(ADR(shapeString),ADR(strHelp));

								x:=smallRadius*COS((angle+36)/180*PI);
								y:=smallRadius*SIN((angle+36)/180*PI);

								strX:=REAL_TO_STRING(x+prevReadX);
								strY:=REAL_TO_STRING(y+prevReadY);
								strHelp:=',';
								strcat(ADR(shapeString),ADR(strX));
								strcat(ADR(shapeString),ADR(strHelp));
								strcat(ADR(shapeString),ADR(strY));
								strHelp:=' ';
								strcat(ADR(shapeString),ADR(strHelp));
								angle:=angle+72;

							END_FOR;

							x:=radius*COS(angle/180*PI);
							y:=radius*SIN(angle/180*PI);
							strX:=REAL_TO_STRING(x+prevReadX);
							strY:=REAL_TO_STRING(y+prevReadY);
							strHelp:=',';
							strcat(ADR(shapeString),ADR(strX));
							strcat(ADR(shapeString),ADR(strHelp));
							strcat(ADR(shapeString),ADR(strY));

							strHelp:='" transform="rotate(';
							strcat(ADR(shapeString),ADR(strHelp));
							strcat(ADR(shapeString),ADR(strRot));
							strHelp:=' ';
							strcat(ADR(shapeString),ADR(strHelp));
							strcat(ADR(shapeString),ADR(strPrevReadX));
							strHelp:=',';
							strcat(ADR(shapeString),ADR(strHelp));
							strcat(ADR(shapeString),ADR(strPrevReadY));
							strHelp:=')"';
							strcat(ADR(shapeString),ADR(strHelp));

							strHelp:='" fill="none" stroke="black" />';
							strcat(ADR(shapeString),ADR(strHelp));
							svgStringArray[svgStringArrayIndex]:=shapeString;

							svgStringArrayIndex:=svgStringArrayIndex+1;

							IF svgStringArray[3]<>'' THEN

								(*PositionArray*)
								strHelp:='type:';
								strcat(ADR(PositionString), ADR(strHelp));
								strcat(ADR(PositionString), ADR(CurrentShape));
								strHelp:='; x=';
								strcat(ADR(PositionString), ADR(strHelp));
								strcat(ADR(PositionString), ADR(strPrevReadX));
								strHelp:='; y=';
								strcat(ADR(PositionString), ADR(strHelp));
								strcat(ADR(PositionString), ADR(strPrevReadY));
								strHelp:='; rot=';
								strcat(ADR(PositionString), ADR(strHelp));
								strcat(ADR(PositionString), ADR(strRot));
								strHelp:='';
								strcat(ADR(PositionString), ADR(strHelp));

								PositionArray[PositionArrayIndex]:=PositionString;
								PositionArrayIndex:=PositionArrayIndex+1;
								PositionString:='';
							END_IF;

							stage:=0;
						END_IF;

					END_IF;
				1:
					InfoString:='Shape outside drawing field!';
					IF EDGEPOS(cmdDraw) THEN
						cmdDraw:=FALSE;
						stage:=0;
					END_IF

				2:
					InfoString:='Distance can not be equal to 0!';
					IF EDGEPOS(cmdDraw) THEN
						cmdDraw:=FALSE;
						stage:=0;
					END_IF;

			END_CASE;

	END_CASE;

(*----clearing paper-----*)
	IF EDGEPOS(cmdClear) THEN
		cmdClear:=FALSE;
		FOR i:=0 TO svgStringArrayIndex DO
			svgStringArray[i]:='';
		END_FOR;
		svgStringArrayIndex:=0;
		FOR i:=0 TO PositionArrayIndex DO
			PositionArray[i]:='';
		END_FOR;
		PositionArrayIndex:=0;
	END_IF;
(*------Undo--------*)
	IF EDGEPOS(cmdBack) THEN
		cmdBack:=FALSE;
		IF svgStringArrayIndex>0 THEN
			svgStringArrayIndex:=svgStringArrayIndex-1;
		END_IF
			svgStringArray[svgStringArrayIndex]:='';

		IF PositionArrayIndex>0 THEN
			PositionArrayIndex:=svgStringArrayIndex-1;
		END_IF
		PositionArray[PositionArrayIndex]:='';
	END_IF;
(*------Pass to global---------*)
	gSvgStringArray:=svgStringArray;
	gSvgStringArrayIndex:=svgStringArrayIndex;

	IF HelpLines THEN

	(* A line showing the position in X*)
	inXlinePosYStr:=REAL_TO_STRING(inXlinePosY);
	inXlinePosXStr:=REAL_TO_STRING(inXlinePosX);
	inXlinePosYStr1:=REAL_TO_STRING(inXlinePosY1);

	gSvgStringArray[0]:='<polyline points="';
	inXlinePosY1:=0;
	strcat(ADR(gSvgStringArray[0]),ADR(inXlinePosXStr));
	strHelp:=',';
	strcat(ADR(gSvgStringArray[0]),ADR(strHelp));
	strcat(ADR(gSvgStringArray[0]),ADR(inXlinePosYStr1));
	strHelp:=' ';
	strcat(ADR(gSvgStringArray[0]),ADR(strHelp));
	inXlinePosY:=630;
	strcat(ADR(gSvgStringArray[0]),ADR(inXlinePosXStr));
	strHelp:=',';
	strcat(ADR(gSvgStringArray[0]),ADR(strHelp));
	strcat(ADR(gSvgStringArray[0]),ADR(inXlinePosYStr));
	strHelp:='" fill="none" stroke="red" />';
	strcat(ADR(gSvgStringArray[0]),ADR(strHelp));

	(* A line showing the position in Y*)
	inYlinePosYStr:=REAL_TO_STRING(inYlinePosY);
	inYlinePosXStr:=REAL_TO_STRING(inYlinePosX);
	inYlinePosXStr1:=REAL_TO_STRING(inYlinePosX1);

	gSvgStringArray[1]:='<polyline points="';
	inYlinePosX1:=0;
	strcat(ADR(gSvgStringArray[1]),ADR(inYlinePosXStr1));
	strHelp:=',';
	strcat(ADR(gSvgStringArray[1]),ADR(strHelp));
	strcat(ADR(gSvgStringArray[1]),ADR(inYlinePosYStr));
	strHelp:=' ';
	strcat(ADR(gSvgStringArray[1]),ADR(strHelp));
	inYlinePosX:=780;
	strcat(ADR(gSvgStringArray[1]),ADR(inYlinePosXStr));
	strHelp:=',';
	strcat(ADR(gSvgStringArray[1]),ADR(strHelp));
	strcat(ADR(gSvgStringArray[1]),ADR(inYlinePosYStr));
	strHelp:='" fill="none" stroke="red" />';
		strcat(ADR(gSvgStringArray[1]),ADR(strHelp));

		(* A circle*)

		gSvgStringArray[2]:='<circle cx="';

		strHelp:='" cy="';
		strcat(ADR(gSvgStringArray[2]),ADR(inXlinePosXStr));
		strcat(ADR(gSvgStringArray[2]),ADR(strHelp));
		strcat(ADR(gSvgStringArray[2]),ADR(inYlinePosYStr));
		strHelp:='" r="20" stroke="red" stroke-width="1" fill="none" />';
		strcat(ADR(gSvgStringArray[2]),ADR(strHelp));
	ELSE
		(* A line showing the position in X*)
		inXlinePosYStr:=REAL_TO_STRING(inXlinePosY);
		inXlinePosXStr:=REAL_TO_STRING(inXlinePosX);
		inXlinePosYStr1:=REAL_TO_STRING(inXlinePosY1);

		gSvgStringArray[0]:='<polyline points="';
		inXlinePosY1:=0;
		strcat(ADR(gSvgStringArray[0]),ADR(inXlinePosXStr));
		strHelp:=',';
		strcat(ADR(gSvgStringArray[0]),ADR(strHelp));
		strcat(ADR(gSvgStringArray[0]),ADR(inXlinePosYStr1));
		strHelp:=' ';
		strcat(ADR(gSvgStringArray[0]),ADR(strHelp));
		inXlinePosY:=630;
		strcat(ADR(gSvgStringArray[0]),ADR(inXlinePosXStr));
		strHelp:=',';
		strcat(ADR(gSvgStringArray[0]),ADR(strHelp));
		strcat(ADR(gSvgStringArray[0]),ADR(inXlinePosYStr));
		strHelp:='" fill="none" stroke="white" />';
		strcat(ADR(gSvgStringArray[0]),ADR(strHelp));

		(* A line showing the position in Y*)
		inYlinePosYStr:=REAL_TO_STRING(inYlinePosY);
		inYlinePosXStr:=REAL_TO_STRING(inYlinePosX);
		inYlinePosXStr1:=REAL_TO_STRING(inYlinePosX1);

		gSvgStringArray[1]:='<polyline points="';
		inYlinePosX1:=0;
		strcat(ADR(gSvgStringArray[1]),ADR(inYlinePosXStr1));
		strHelp:=',';
		strcat(ADR(gSvgStringArray[1]),ADR(strHelp));
		strcat(ADR(gSvgStringArray[1]),ADR(inYlinePosYStr));
		strHelp:=' ';
		strcat(ADR(gSvgStringArray[1]),ADR(strHelp));
		inYlinePosX:=780;
		strcat(ADR(gSvgStringArray[1]),ADR(inYlinePosXStr));
		strHelp:=',';
		strcat(ADR(gSvgStringArray[1]),ADR(strHelp));
		strcat(ADR(gSvgStringArray[1]),ADR(inYlinePosYStr));
		strHelp:='" fill="none" stroke="white" />';
		strcat(ADR(gSvgStringArray[1]),ADR(strHelp));

		(* A circle*)

		gSvgStringArray[2]:='<circle cx="';

		strHelp:='" cy="';
		strcat(ADR(gSvgStringArray[2]),ADR(inXlinePosXStr));
		strcat(ADR(gSvgStringArray[2]),ADR(strHelp));
		strcat(ADR(gSvgStringArray[2]),ADR(inYlinePosYStr));
		strHelp:='" r="20" stroke="white" stroke-width="2" fill="none" />';
		strcat(ADR(gSvgStringArray[2]),ADR(strHelp));
	END_IF;

END_PROGRAM

PROGRAM _EXIT
	(* Insert code here *)

END_PROGRAM
```

### Program Logical/Programs/live_drawing/svg_to_gcode

#### Variables.var
```iecst
VAR
	j : UINT;
	i : UINT;
	svgString : STRING[500];
	labelString : STRING[80];
	flag1 : BOOL;
	buff : STRING[80];
	xory : BOOL;
	strDevice : STRING[80];
	strFile : STRING[80];
	FCreate : FileCreate;
	FClose : FileClose;
	cncString : STRING[100000];
	FWrite : FileWrite;
	cmdFile : BOOL;
	FOpen : FileOpen;
	byStep : INT;
	bOK : BOOL;
	byErrorLevel : INT;
	dwIdent : UDINT;
	wStatus : UINT;
	wError : UINT;
	strHelp : STRING[80];
	Xstr : STRING[80];
	Ystr : STRING[80];
	Fstr : STRING[80] := '2000';
	cmdConvert : BOOL;
	firstMove : BOOL;
	prevXstr : STRING[80];
	prevYstr : STRING[80];
END_VAR
VAR RETAIN
	fileIndex : INT;
END_VAR
VAR
	strNum : STRING[80];
	k : INT;
	Rstr : STRING[80];
	Xstr2 : STRING[80];
	Ystr2 : STRING[80];
	fileFlag : BOOL;
	Xscale : REAL;
	Yscale : REAL;
	Rscale : REAL;
	Y2scale : REAL;
	X2scale : REAL;
	gMsgBox5 : BOOL;
END_VAR
```

#### Main.st
```iecst
PROGRAM _INIT
	(* Insert code here *)
	strDevice:= 'CNC_PrgDir';
	strFile:= 'obrazek.cnc';
	bOK := FALSE;
	byStep := 1;
	byErrorLevel := 0;

	memset(ADR(cncString), 0, SIZEOF(cncString));
END_PROGRAM

PROGRAM _CYCLIC
	(* Insert code here *)

	IF EDGEPOS(cmdConvert) THEN
		gMsgBox5:=TRUE;
	ELSE
		gMsgBox5:=FALSE;
	END_IF;

	IF cmdConvert THEN

		IF gSvgStringArray[3]<>'' THEN

			memset(ADR(cncString), 0, SIZEOF(cncString));
			strHelp:='%001$n';
			strcat(ADR(cncString),ADR(strHelp));
			FOR i:=3 TO (gSvgStringArrayIndex-1) DO

				svgString:=gSvgStringArray[i];
				labelString:=LEFT(svgString,4);
				Xstr:='';
				Ystr:='';
				Rstr:='';
				IF labelString='<pol' THEN
					j:=19;
					flag1:=TRUE;
					firstMove:=TRUE;
					WHILE flag1 DO
						buff:=MID(svgString,1,j);

						IF buff=',' THEN
							xory:=TRUE;

						ELSIF buff=' ' OR buff='"' THEN
							xory:=FALSE;

							Xscale:=STRING_TO_REAL(Xstr)/1.5;
							Xstr:=REAL_TO_STRING(Xscale);
							Yscale:=STRING_TO_REAL(Ystr)/1.5;
							Ystr:=REAL_TO_STRING(Yscale);

							IF firstMove THEN
								IF prevXstr<>Xstr OR prevYstr<>Ystr THEN
									strHelp:='M50$n';    //podniesienie

									strcat(ADR(cncString),ADR(strHelp));

									strHelp:='G01 X';
									strcat(ADR(cncString),ADR(strHelp));
									strcat(ADR(cncString),ADR(Xstr));
									strHelp:=' Z';
									strcat(ADR(cncString),ADR(strHelp));
									strcat(ADR(cncString),ADR(Ystr));
									strHelp:=' F';
									strcat(ADR(cncString),ADR(strHelp));
									strcat(ADR(cncString),ADR(Fstr));
									strHelp:='$n';
									strcat(ADR(cncString),ADR(strHelp));

									strHelp:='M60$n';    //opuszczenie

									strcat(ADR(cncString),ADR(strHelp));
								END_IF
								firstMove:=FALSE;
							ELSE
								strHelp:='G01 X';
								strcat(ADR(cncString),ADR(strHelp));
								strcat(ADR(cncString),ADR(Xstr));
								strHelp:=' Z';
								strcat(ADR(cncString),ADR(strHelp));
								strcat(ADR(cncString),ADR(Ystr));
								strHelp:=' F';
								strcat(ADR(cncString),ADR(strHelp));
								strcat(ADR(cncString),ADR(Fstr));
								strHelp:='$n';
								strcat(ADR(cncString),ADR(strHelp));
							END_IF

							prevXstr:=Xstr;
							prevYstr:=Ystr;

							Xstr:='';
							Ystr:='';

							IF buff='"' THEN
								flag1:=FALSE;
							END_IF

						ELSE
							IF xory THEN
								strcat(ADR(Ystr),ADR(buff));
							ELSE

								strcat(ADR(Xstr),ADR(buff));
							END_IF
						END_IF
						j:=j+1;
					END_WHILE;

				ELSIF labelString='<cir' THEN
					j:=12;
					flag1:=TRUE;
					k:=0;
					WHILE flag1 DO
						buff:=MID(svgString,1,j);

						IF buff='"' THEN

							k:=k+1;
						ELSE

							CASE k OF
								1:

									strcat(ADR(Xstr),ADR(buff));
								3:
									strcat(ADR(Ystr),ADR(buff));
								5:
									strcat(ADR(Rstr),ADR(buff));
								6:	flag1:=FALSE;
									strHelp:='M50$n';    //podniesienie
									Xscale:=STRING_TO_REAL(Xstr)/1.5;
									Xstr:=REAL_TO_STRING(Xscale);
									Yscale:=STRING_TO_REAL(Ystr)/1.5;
									Ystr:=REAL_TO_STRING(Yscale);
									Rscale:=STRING_TO_REAL(Rstr)/1.5;
									Rstr:=REAL_TO_STRING(Rscale);

									Xstr:=REAL_TO_STRING(STRING_TO_REAL(Xstr)-STRING_TO_REAL(Rstr));

									strcat(ADR(cncString),ADR(strHelp));
									strHelp:='G01 X';
									strcat(ADR(cncString),ADR(strHelp));
									strcat(ADR(cncString),ADR(Xstr));
									strHelp:=' Z';
									strcat(ADR(cncString),ADR(strHelp));
									strcat(ADR(cncString),ADR(Ystr));
									strHelp:=' F';
									strcat(ADR(cncString),ADR(strHelp));
									strcat(ADR(cncString),ADR(Fstr));
									strHelp:='$n';
									strcat(ADR(cncString),ADR(strHelp));
									strHelp:='M60$n';    //opuszczenie
									strcat(ADR(cncString),ADR(strHelp));
									strHelp:='G02 I';
									strcat(ADR(cncString),ADR(strHelp));
									strcat(ADR(cncString),ADR(Rstr));
									strHelp:=' H360$n';
									strcat(ADR(cncString),ADR(strHelp));
									Xstr:='';
									Ystr:='';
									Rstr:='';

							END_CASE;
						END_IF

						j:=j+1;
					END_WHILE;

				ELSIF labelString='<pat' THEN
					j:=11;
					flag1:=TRUE;
					k:=0;
					WHILE flag1 DO
						buff:=MID(svgString,1,j);

						IF buff=' ' THEN

							k:=k+1;

						ELSIF buff='"' THEN
							flag1:=FALSE;
							Xscale:=STRING_TO_REAL(Xstr)/1.5;
							Xstr:=REAL_TO_STRING(Xscale);
							Yscale:=STRING_TO_REAL(Ystr)/1.5;
							Ystr:=REAL_TO_STRING(Yscale);

							X2scale:=STRING_TO_REAL(Xstr2)/1.5;
							Xstr2:=REAL_TO_STRING(X2scale);
							Y2scale:=STRING_TO_REAL(Ystr2)/1.5;
							Ystr2:=REAL_TO_STRING(Y2scale);

							Rscale:=STRING_TO_REAL(Rstr)/1.5;
							Rstr:=REAL_TO_STRING(Rscale);
							IF prevXstr<>Xstr OR prevYstr<>Ystr THEN
								strHelp:='M50$n';    //podniesienie

								strcat(ADR(cncString),ADR(strHelp));
								strHelp:='G01 X';
								strcat(ADR(cncString),ADR(strHelp));
								strcat(ADR(cncString),ADR(Xstr));
								strHelp:=' Z';
								strcat(ADR(cncString),ADR(strHelp));
								strcat(ADR(cncString),ADR(Ystr));
								strHelp:=' F';
								strcat(ADR(cncString),ADR(strHelp));
								strcat(ADR(cncString),ADR(Fstr));
								strHelp:='$n';
								strcat(ADR(cncString),ADR(strHelp));
								strHelp:='M60$n';    //opuszczenie
								strcat(ADR(cncString),ADR(strHelp));

							END_IF

							strHelp:='G03 X';
							strcat(ADR(cncString),ADR(strHelp));
							strcat(ADR(cncString),ADR(Xstr2));
							strHelp:=' Z';
							strcat(ADR(cncString),ADR(strHelp));
							strcat(ADR(cncString),ADR(Ystr2));
							strHelp:=' R=';
							strcat(ADR(cncString),ADR(strHelp));
							strcat(ADR(cncString),ADR(Rstr));
							strHelp:='$n';
							strcat(ADR(cncString),ADR(strHelp));
							prevXstr:=Xstr2;
							prevYstr:=Ystr2;

							Xstr:='';
							Ystr:='';
							Rstr:='';
							Xstr2:='';
							Ystr2:='';

						ELSE

							CASE k OF
								1:

									strcat(ADR(Xstr),ADR(buff));
								2:
									strcat(ADR(Ystr),ADR(buff));
								4:
									strcat(ADR(Rstr),ADR(buff));
								9:	strcat(ADR(Xstr2),ADR(buff));

								10:	strcat(ADR(Ystr2),ADR(buff));

							END_CASE;
						END_IF

						j:=j+1;
					END_WHILE;
				END_IF;

			END_FOR;
			strHelp:='M30';
			strcat(ADR(cncString),ADR(strHelp));
			cmdFile:=TRUE;
		END_IF;
		cmdConvert:=FALSE;
	END_IF

	IF cmdFile THEN

		CASE byStep OF
			0: (**** Error step ****)                bOK := FALSE;
			1: (**** Try to open existing file ****)
				(* Initialize file open structrue *)
				FOpen.enable    := 1;
				FOpen.pDevice   := ADR(strDevice);
				FOpen.pFile     := ADR(strFile);
				FOpen.mode      := FILE_RW;  (* Read and write access *)
				(* Call FBK *)                FOpen();
				(* Get FBK output information *)
				dwIdent := FOpen.ident;                wStatus := FOpen.status;
				(* Verify status (20708 -> File doesn't exist) *)
				IF (wStatus = 20708) THEN
					byStep := 2;
					fileFlag:=FALSE;
				ELSE                        IF (wStatus = 0) THEN
						byStep := 5;
						fileFlag:=TRUE;
					ELSE
						IF (wStatus <> 65535) THEN
							byErrorLevel := 1;
							byStep := 0;
							IF (wStatus = 20799) THEN
								wError := FileIoGetSysError();
							END_IF
					END_IF                        END_IF
				END_IF
			2: (**** Create file ****)
				(* Initialize file create structure *)
				FCreate.enable  := 1;
				FCreate.pDevice := ADR(strDevice);
				FCreate.pFile   := ADR(strFile);                (* Call FBK *)
				FCreate();                (* Get FBK output information *)
				dwIdent := FCreate.ident;
				wStatus := FCreate.status;                (* Verify status *)
				IF (wStatus = 0) THEN                        byStep := 3;
				ELSE                        IF (wStatus <> 65535) THEN
						byErrorLevel := 2;
						byStep := 0;
						IF (wStatus = 20799) THEN
							wError := FileIoGetSysError();
					END_IF                        END_IF
				END_IF
			3: (**** Write data to file ****)
				(* Initialize file write structure *)
				FWrite.enable   := 1;               FWrite.ident    := dwIdent;
				FWrite.offset   := 0;
				FWrite.pSrc     := ADR(cncString);
				FWrite.len      := LEN(cncString);
				(* Call FBK *)                FWrite();

				(* Get status *)                wStatus := FWrite.status;
				(* Verify status *)                IF (wStatus = 0) THEN
				byStep := 5;                ELSE
					IF (wStatus <> 65535) THEN
						byErrorLevel := 3;
						byStep := 0;
						IF (wStatus = 20799) THEN
							wError := FileIoGetSysError();
					END_IF                        END_IF
				END_IF
				//		4: (**** Read data from file ****)
				//			(* Initialize file read structure *)
				//			FRead.enable    := 1;                FRead.ident     := dwIdent;
				//			FRead.offset    := 0;
				//			FRead.pDest     := ADR(byReadData[0]);
				//			FRead.len       := SIZEOF(byReadData);
				//			(* Call FBK *)                FRead();
				//			(* Get status *)                wStatus := FRead.status;
				//			(* Verify status *)                IF (wStatus = 0) THEN
				//			byStep := 5;                ELSE
				//				IF (wStatus <> 65535) THEN
				//					byErrorLevel := 4;
				//					byStep := 0;
				//					IF (wStatus = 20799) THEN
				//						wError := FileIoGetSysError();
				//				END_IF                        END_IF
				//			END_IF
			5: (**** Close file ****)
				(* Initialize file close structure *)
				FClose.enable   := 1;                FClose.ident    := dwIdent;
				(* Call FBK *)                FClose();
				(* Get status *)                wStatus := FClose.status;
				(* Verify status *)
				IF (wStatus = 0) THEN

					IF fileFlag THEN

					ELSE

						cmdFile:=FALSE;
						memset(ADR(cncString), 0, SIZEOF(cncString));
					END_IF
					byStep := 1;
					fileIndex:=fileIndex+1;
					strNum:=INT_TO_STRING(fileIndex);
					strFile:='obrazek.cnc';
					strFile := INSERT(strFile, strNum, 7);

				ELSE
					IF (wStatus <> 65535) THEN
						byErrorLevel := 5;
						byStep := 0;

						IF (wStatus = 20799) THEN
							wError := FileIoGetSysError();
					END_IF                        END_IF
				END_IF
			//		6: (**** Delete file ****)
			//			(* Initialize file delete structure *)
			//			FDelete.enable  := 1;
			//			FDelete.pDevice := ADR(strDevice);
			//			FDelete.pName   := ADR(strFile);                (* Call FBK *)
			//			FDelete();                (* Get status *)
			//			wStatus := FDelete.status;                (* Verify status *)
			//			IF (wStatus = 0) THEN                        bOK     := TRUE;
			//			byStep := 7;                ELSE
			//				IF (wStatus <> 65535) THEN
			//					byErrorLevel := 6;
			//					byStep := 0;
			//					IF (wStatus = 20799) THEN
			//						wError := FileIoGetSysError();
			//					END_IF
			//				END_IF
			//			END_IF
		END_CASE

	END_IF

END_PROGRAM

PROGRAM _EXIT
	(* Insert code here *)

END_PROGRAM
```

### Program Logical/Programs/Recipe (IEC)

#### Variables.var
```iecst
VAR
	i : UINT;
	j : UINT;
	k : INT;
	MpRecipeRegPar_0 : MpRecipeRegPar;
	MpRecipeUI_0 : MpRecipeUI;
	MpRecipeXml_0 : MpRecipeXml;
	nextAddr : UDINT;
	TempLine : ARRAY[0..4] OF STRING[80];
	UIConnect : MpRecipeUIConnectType := (Recipe:=(SortOrder:=mpRECIPE_UI_SORT_DATE_ASCENDING));
	UISetup : MpRecipeUISetupType := (RecipeListSize:=20);
	DataProvider0 : ARRAY[0..4] OF STRING[100];
	CreatingRecipe : BOOL;
END_VAR
```

#### ConnectWordsAction.st
```iecst
ACTION ConnectWords:

	FOR k:=0 TO 4 DO
		memset(ADR(TempLine[k]),0,SIZEOF(TempLine[k]));
		memset(ADR(DataProvider0[k]),0, SIZEOF(DataProvider0[k]));
	END_FOR;

	FOR i:=0 TO 4 DO
		TempLine[0]:='{"value":"';
		TempLine[1]:=INT_TO_STRING(i);
		TempLine[2]:='","text":"';
		TempLine[3]:=UIConnect.Recipe.List.Names[i];
		TempLine[4]:='"}';

		nextAddr:=strcat(ADR(DataProvider0[i]), ADR(TempLine[0]));

		FOR j:=1 TO 4 DO
			strcat(nextAddr,ADR(TempLine[j]));
		END_FOR;

	END_FOR;

END_ACTION
```

#### Main.st
```iecst
PROGRAM _INIT

END_PROGRAM

PROGRAM _CYCLIC

	// basic settings for recipes
	MpRecipeXml_0(MpLink:= ADR(gRecipeXml), Enable := TRUE, DeviceName := ADR('CF'), FileName := ADR('recipe') );

	MpRecipeRegPar_0(MpLink:= ADR(gRecipeXml), Enable := TRUE, PVName := ADR('gParameter') );

	MpRecipeUI_0(MpLink:= ADR(gRecipeXml), Enable := TRUE, UISetup := UISetup, UIConnect := ADR(UIConnect));

	UIConnect.Recipe.Filter:='*.xml';

	ConnectWords;
	MaxNumOfRecipes;

END_PROGRAM

PROGRAM _EXIT

	MpRecipeXml_0.Save:= TRUE;
	MpRecipeXml_0.Enable:=FALSE;
	MpRecipeXml_0();

	MpRecipeRegPar_0.Enable:=FALSE;
	MpRecipeRegPar_0();

END_PROGRAM
```

#### MessageBoxAction.st
```iecst
ACTION MaxNumOfRecipes:

	// Messagebox informs that the maximum number of recipes has been reached
	IF UIConnect.Recipe.List.MaxSelection>=5 AND CreatingRecipe  THEN
		gMsgBox4:=TRUE;
		CreatingRecipe := FALSE;
	END_IF;

END_ACTION
```

### Variables.var
```iecst
VAR

	toolUp : BOOL;
	toolDown : BOOL;

	DialogErrorVisible : BOOL;

	MC_BR_MFunction_0 : MC_BR_MFunction;
	MC_BR_MFunction_1 : MC_BR_MFunction;

END_VAR
```

### Program Logical/Programs/UserManagement/UsrMgmtP

#### Variables.var
```iecst
VAR
	LabelFirstLoginVisible : BOOL;
	DateFirstLoginVisible : BOOL;
	StringError : WSTRING[80];
	EditUserRoleIndex : USINT;
	NewUserRoleIndex : USINT;
	DialogEditUserConfirmEnabled : BOOL;
	DialogNewUserConfirmEnabled : BOOL;
	SelectedUser : WSTRING[80];
	EditUserPasswordOk : WSTRING[80];
	NewUserPasswordOk : WSTRING[80];
	SelectedUserGroup : WSTRING[80];
	LoggedAs : WSTRING[80];
	EditUserPasswordHint : WSTRING[80];
	NewUserPasswordHint : WSTRING[80];
	MpUserXLoginUIConnect0 : MpUserXLoginUIConnectType;
	MpUserXLoginUI_0 : MpUserXLoginUI;
	MpUserXMgrUIConnect_0 : MpUserXMgrUIConnectType;
	MpUserXLogin_0 : MpUserXLogin;
	MpUserXManagerUI_0 : MpUserXManagerUI;
	MpUserXMgrUISetup_0 : MpUserXMgrUISetupType;
END_VAR
```

#### Main.st
```iecst
PROGRAM _INIT

	MpUserXLogin_0.Enable := 1;
	MpUserXLogin_0.MpLink := ADR(gUserXLogin);

	MpUserXManagerUI_0.Enable := 1;
	MpUserXManagerUI_0.MpLink := ADR(gUserXLogin);
	MpUserXManagerUI_0.UIConnect := ADR(MpUserXMgrUIConnect_0);
	MpUserXManagerUI_0.UISetup := MpUserXMgrUISetup_0;

	MpUserXLoginUI_0.Enable := 1;
	MpUserXLoginUI_0.MpLink := ADR(gUserXLogin);
	MpUserXLoginUI_0.UIConnect := ADR(MpUserXLoginUIConnect0);

END_PROGRAM

PROGRAM _CYCLIC

	//DISPLAY SELECTED USER
	SelectedUser := MpUserXMgrUIConnect_0.User.List.UserNames[MpUserXMgrUIConnect_0.User.List.SelectedIndex];

	//USER GROUPS DISPLAY
	CASE MpUserXMgrUIConnect_0.User.Info.Roles[0] OF
		1:
			SelectedUserGroup := "Administrator";
		2:
			SelectedUserGroup := "Anonymous";
		3:
			SelectedUserGroup := "Operator";
	END_CASE;

	//NEW USER ROLE
	MpUserXMgrUIConnect_0.User.Create.Dialog.Roles[0] := NewUserRoleIndex + 2;

	//EDITING USER ROLE
	MpUserXMgrUIConnect_0.User.Edit.Dialog.Roles[0] := EditUserRoleIndex + 2;

	//FUNCTION CALL
	MpUserXLogin_0();
	MpUserXLoginUI_0();
	MpUserXManagerUI_0();

END_PROGRAM

PROGRAM _EXIT

	MpUserXLogin_0.Enable := 0;
	MpUserXLogin_0();

	MpUserXLoginUI_0.Enable := 0;
	MpUserXLoginUI_0();

	MpUserXManagerUI_0.Enable := 0;
	MpUserXManagerUI_0();

END_PROGRAM
```

### Program Logical/Programs/UsrMgmtP (IEC)

#### Main.st - Init, cyclic, exit code
```iecst
PROGRAM _INIT

	MpUserXLogin_0.Enable := 1;
	MpUserXLogin_0.MpLink := ADR(gUserXLogin);

	MpUserXManagerUI_0.Enable := 1;
	MpUserXManagerUI_0.MpLink := ADR(gUserXLogin);
	MpUserXManagerUI_0.UIConnect := ADR(MpUserXMgrUIConnect_0);
	MpUserXManagerUI_0.UISetup := MpUserXMgrUISetup_0;

	MpUserXLoginUI_0.Enable := 1;
	MpUserXLoginUI_0.MpLink := ADR(gUserXLogin);
	MpUserXLoginUI_0.UIConnect := ADR(MpUserXLoginUIConnect0);

END_PROGRAM

PROGRAM _CYCLIC

	//DISPLAY SELECTED USER
	SelectedUser := MpUserXMgrUIConnect_0.User.List.UserNames[MpUserXMgrUIConnect_0.User.List.SelectedIndex];

	//USER GROUPS DISPLAY
	CASE MpUserXMgrUIConnect_0.User.Info.Roles[0] OF
		1:
			SelectedUserGroup := "Administrator";
		2:
			SelectedUserGroup := "Anonymous";
		3:
			SelectedUserGroup := "Operator";
	END_CASE;

	//NEW USER ROLE
	MpUserXMgrUIConnect_0.User.Create.Dialog.Roles[0] := NewUserRoleIndex + 2;

	//EDITING USER ROLE
	MpUserXMgrUIConnect_0.User.Edit.Dialog.Roles[0] := EditUserRoleIndex + 2;

	//FUNCTION CALL
	MpUserXLogin_0();
	MpUserXLoginUI_0();
	MpUserXManagerUI_0();

	VisuAction;
END_PROGRAM

PROGRAM _EXIT

	MpUserXLogin_0.Enable := 0;
	MpUserXLogin_0();

	MpUserXLoginUI_0.Enable := 0;
	MpUserXLoginUI_0();

	MpUserXManagerUI_0.Enable := 0;
	MpUserXManagerUI_0();

END_PROGRAM
```

#### Variables.var - Local variables
```iecst
VAR
	EditUserRoleIndex : USINT;
	NewUserRoleIndex : USINT;
	SelectedUser : WSTRING[80];
	SelectedUserGroup : WSTRING[80];
	MpUserXLoginUIConnect0 : MpUserXLoginUIConnectType;
	MpUserXLoginUI_0 : MpUserXLoginUI;
	MpUserXMgrUIConnect_0 : MpUserXMgrUIConnectType;
	MpUserXLogin_0 : MpUserXLogin;
	MpUserXManagerUI_0 : MpUserXManagerUI;
	MpUserXMgrUISetup_0 : MpUserXMgrUISetupType;
END_VAR
```

#### Action.st
```iecst
ACTION VisuAction:
	Show;
	NumericInput;
	SliderInput;
END_ACTION
```

- Project.language (not shown)

### Program Logical/CNC_FMU

#### Variables.var
```iecst
VAR
	MC_ReadActualTorque_0 : MC_ReadActualTorque;
	MC_ReadActualTorque_1 : MC_ReadActualTorque;
	CNC_FMU1 : CNC_FMU;
	CNC_FMUView_0 : CNC_FMUView;
	MC_BR_WrLoadSimPosition_AcpAx_0 : MC_BR_WrLoadSimPosition_AcpAx;
	MC_BR_WrLoadSimPosition_AcpAx_1 : MC_BR_WrLoadSimPosition_AcpAx;
END_VAR
```

#### Main.st
```iecst
PROGRAM _INIT

	MC_BR_WrLoadSimPosition_AcpAx_0.Axis:=ADR(gAxisQX);
	MC_BR_WrLoadSimPosition_AcpAx_1.Axis:=ADR(gAxisQZ);

	MC_ReadActualTorque_0.Axis:=ADR(gAxisQX);
	MC_ReadActualTorque_1.Axis:=ADR(gAxisQZ);

	MC_ReadActualTorque_0.Enable:=TRUE;
	MC_ReadActualTorque_1.Enable:=TRUE;

	CNC_FMU1.Enable:=TRUE;
	CNC_FMUView_0.Enable:=TRUE;

END_PROGRAM

PROGRAM _CYCLIC

	MC_BR_WrLoadSimPosition_AcpAx_0.Enable:=MpAxisBasicX.Info.ReadyToPowerOn;
	MC_BR_WrLoadSimPosition_AcpAx_1.Enable:=MpAxisBasicY.Info.ReadyToPowerOn;

	MC_ReadActualTorque_0();
	MC_ReadActualTorque_1();

	CNC_FMU1.X:=MC_ReadActualTorque_0.Torque;
	CNC_FMU1.Y:=MC_ReadActualTorque_1.Torque;

	CNC_FMU1();

	MC_BR_WrLoadSimPosition_AcpAx_0.Position:=CNC_FMU1.PositionX;
	MC_BR_WrLoadSimPosition_AcpAx_1.Position:=CNC_FMU1.PositionY;

	MC_BR_WrLoadSimPosition_AcpAx_0();
	MC_BR_WrLoadSimPosition_AcpAx_1();

	CNC_FMUView_0.InstRef:=CNC_FMU1.InstRef;

	CNC_FMUView_0();

END_PROGRAM

PROGRAM _EXIT
	(* Insert code here *)

END_PROGRAM
```

### Library Logical/CNC_FMUFmu2/CNC_FMULib (ANSIC)
Depends on: sys_lib

#### Types.typ - Exported data types
```iecst
TYPE
	CNC_FMULibFmi2CbType : 	STRUCT
		Logger : UDINT;
		AllocateMemory : UDINT;
		FreeMemory : UDINT;
		StepFinished : UDINT;
		ComponentEnvironment : UDINT;
	END_STRUCT;
	CNC_FMULibFmi2IfType : 	STRUCT
		Enabled : BOOL;
		StartTime : LREAL;
		EndTime : LREAL;
		CurrentTime : LREAL;
		StepSize : LREAL;
		Error : DINT;
		Instance : UDINT;
		Callbacks : CNC_FMULibFmi2CbType;
	END_STRUCT;
	CNC_FMUInternalType : 	STRUCT
		Fmi2 : CNC_FMULibFmi2IfType;
	END_STRUCT;
END_TYPE
```

#### CNC_FMULib.fun - Exported functions and function blocks
```iecst
FUNCTION_BLOCK CNC_FMUView
	VAR_INPUT
		Enable : BOOL;
		InstRef : REFERENCE TO CNC_FMUInternalType;
	END_VAR
	VAR_OUTPUT
		ObjPos : ARRAY[0..18] OF REAL;
	END_VAR
	VAR
		vInternal : ARRAY[0..18] OF LREAL;
	END_VAR
END_FUNCTION_BLOCK

FUNCTION_BLOCK CNC_FMU (**) (*$GROUP=User,$CAT=User,$GROUPICON=User.png,$CATICON=User.png*) (*Fmu.Type="CNC_FMU",Fmu.ModelName="CNC_FMU",Fmu.GUID="{0f3398f8-206d-0d3a-c8cf-c7c7b11e43f1}",Fmu.LocalPath="C:\Users\VOSTRO 5000 Series\Desktop\CNC_FMU.fmu",Fmu.Updated="2021-01-25 13:39:10"*)
	VAR_INPUT
		Enable : BOOL;
	END_VAR
	VAR_OUTPUT
		InstRef : UDINT;
	END_VAR
	VAR
		Internal : CNC_FMUInternalType;
	END_VAR
	VAR_INPUT
		X : LREAL; (*X*)
		Y : LREAL; (*Y*)
	END_VAR
	VAR_OUTPUT
		PositionX : LREAL; (*PositionX*)
		PositionY : LREAL; (*PositionY*)
		SpeedX : LREAL; (*der(P1.s)*)
		SpeedY : LREAL; (*der(P2.s)*)
		TorqueX : LREAL; (*TorqueX*)
		TorqueY : LREAL; (*TorqueY*)
	END_VAR
END_FUNCTION_BLOCK
```
